% RSLogix 500 project M8017 SEALER OVEN B 20170728 CBP.RSS, saved by version 8.30.00.16 %
PROJECT "M8017"    % processor: MicroLogix 1200 %

PROGRAM FILES
  LAD 2 "MAIN_PROG"  15 rungs
  LAD 4 "INF_XFR_IO"  9 rungs  % InFeed Transfer Input / Output %
  LAD 5 "INF_LOAD"  22 rungs  % InFeed Load Cycle %
  LAD 6 "LANES"  15 rungs  % Lane Conveyor Control %
  LAD 7 "OUT_XFR_IO"  15 rungs  % OutFeed Transfer Input / Output %
  LAD 8 "OUT_UNLOAD"  20 rungs  % OutFeed UnLoad Cycle %
  LAD 10 "FLT"  4 rungs  % Operation Faults %
  LAD 11 "PTV"  8 rungs
  LAD 12 "TOP COAT B"  21 rungs

DATA FILES
  O0 OUTPUT  5 elements
  I1 INPUT  6 elements
  S2 STATUS  66 elements
  B3 BINARY  100 elements
  T4 TIMER  90 elements
  C5 COUNTER  6 elements
  R6 CONTROL  6 elements
  N7 INTEGER  81 elements
  F8 FLOAT  1 elements
  B9 OSR_BIT_2  10 elements  % One Shot Relays and Bit Level 2 %
  B10 HMI  10 elements
  MG11 C8014  1 elements
  T41 TMR_2  100 elements  % Timer Level 2 %
  N71 INT_2  100 elements  % Integer Level 2 %

LADDER 2 "MAIN_PROG"
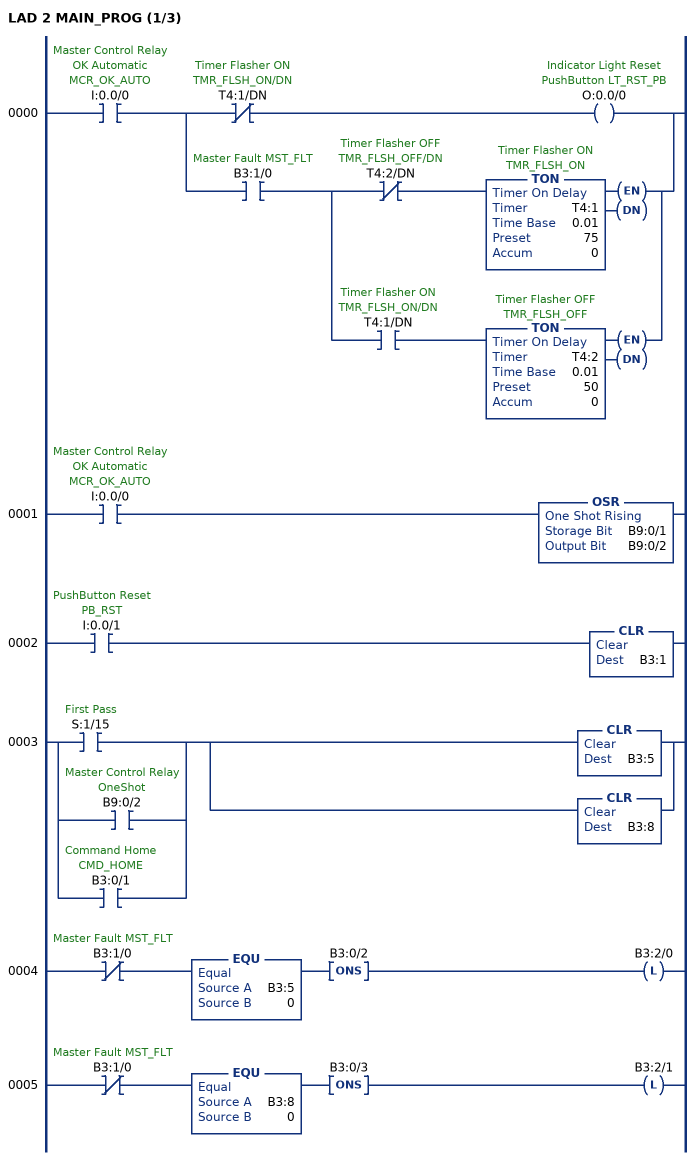
% Rung: 0 %
SOR XIC I:0.0/0 BST XIO T4:1/DN OTE O:0.0/0 NXB XIC B3:1/0 BST XIO T4:2/DN TON T4:1 0.01 75 0 NXB XIC T4:1/DN TON T4:2 0.01 50 0 BND BND EOR
%   I:0.0/0  MCR_OK_AUTO  "Master Control Relay OK Automatic" %
%   T4:1  TMR_FLSH_ON  "Timer Flasher ON" %
%   O:0.0/0  LT_RST_PB  "Indicator Light Reset PushButton" %
%   B3:1/0  MST_FLT  "Master Fault" %
%   T4:2  TMR_FLSH_OFF  "Timer Flasher OFF" %
% Rung: 1 %
SOR XIC I:0.0/0 OSR B9:0/1 B9:0/2 EOR
%   I:0.0/0  MCR_OK_AUTO  "Master Control Relay OK Automatic" %
%   B9:0/2  "Master Control Relay OneShot" %
% Rung: 2 %
SOR XIC I:0.0/1 CLR B3:1 EOR
%   I:0.0/1  PB_RST  "PushButton Reset" %
% Rung: 3 %
SOR BST XIC S:1/15 NXB XIC B9:0/2 NXB XIC B3:0/1 BND BST CLR B3:5 NXB CLR B3:8 BND EOR
%   S:1/15  "First Pass" %
%   B9:0/2  "Master Control Relay OneShot" %
%   B3:0/1  CMD_HOME  "Command Home" %
% Rung: 4 %
SOR XIO B3:1/0 EQU B3:5 0 ONS B3:0/2 OTL B3:2/0 EOR
%   B3:1/0  MST_FLT  "Master Fault" %
% Rung: 5 %
SOR XIO B3:1/0 EQU B3:8 0 ONS B3:0/3 OTL B3:2/1 EOR
%   B3:1/0  MST_FLT  "Master Fault" %

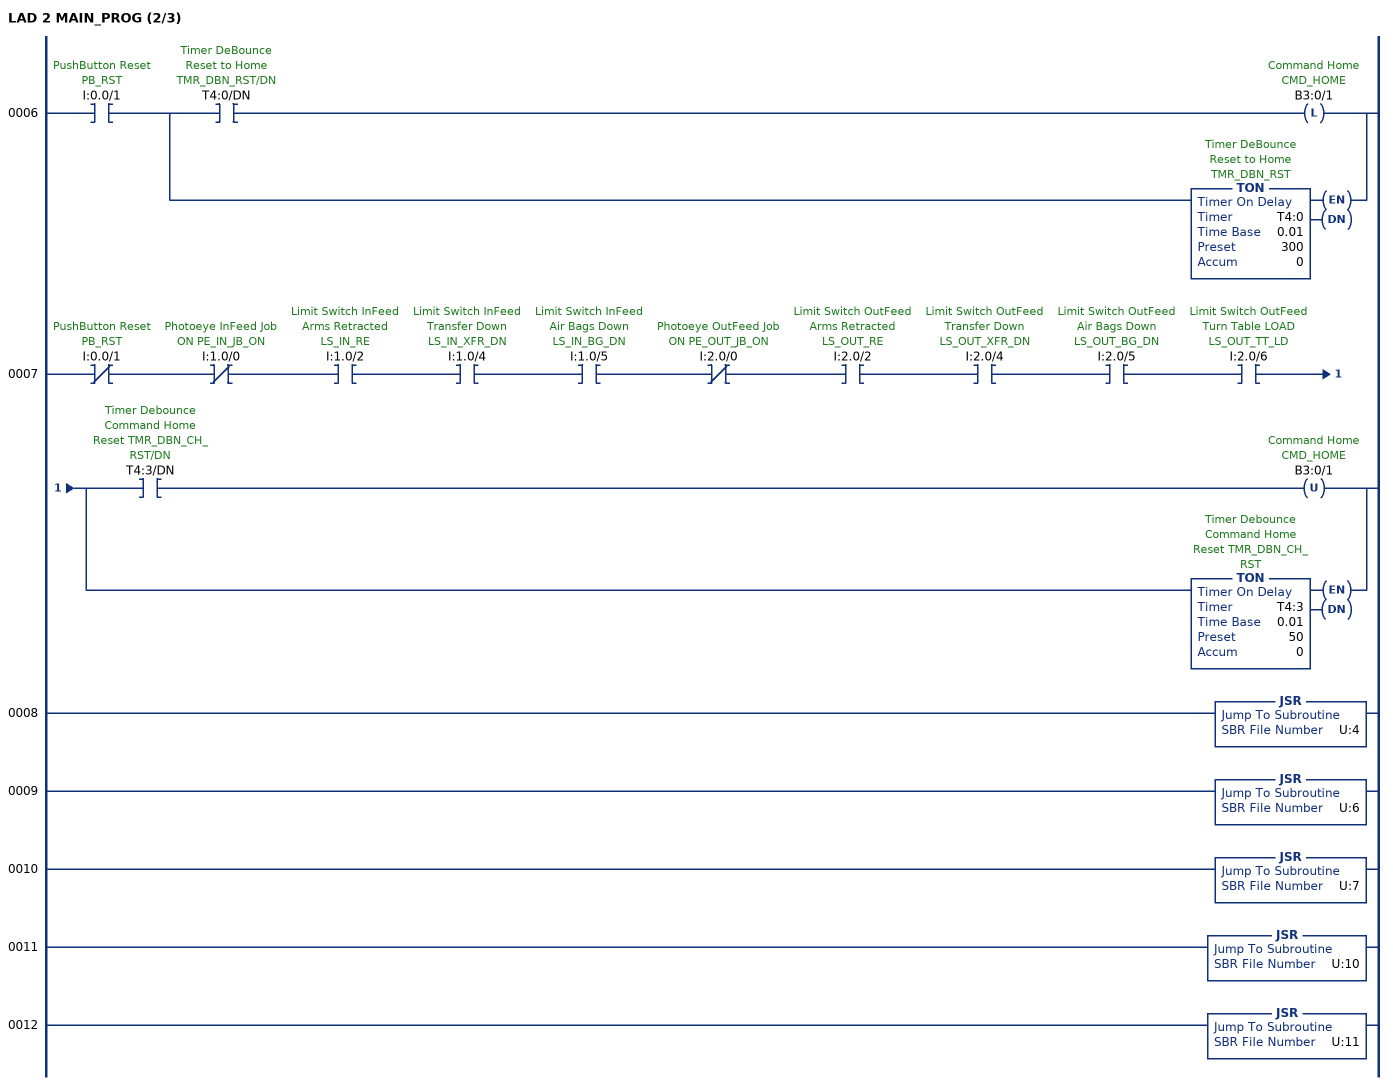
% Rung: 6 %
SOR XIC I:0.0/1 BST XIC T4:0/DN OTL B3:0/1 NXB TON T4:0 0.01 300 0 BND EOR
%   I:0.0/1  PB_RST  "PushButton Reset" %
%   T4:0  TMR_DBN_RST  "Timer DeBounce Reset to Home" %
%   B3:0/1  CMD_HOME  "Command Home" %
% Rung: 7 %
SOR XIO I:0.0/1 XIO I:1.0/0 XIC I:1.0/2 XIC I:1.0/4 XIC I:1.0/5 XIO I:2.0/0 XIC I:2.0/2 XIC I:2.0/4 XIC I:2.0/5 XIC I:2.0/6 BST XIC T4:3/DN OTU B3:0/1 NXB TON T4:3 0.01 50 0 BND EOR
%   I:0.0/1  PB_RST  "PushButton Reset" %
%   I:1.0/0  PE_IN_JB_ON  "Photoeye InFeed Job ON" %
%   I:1.0/2  LS_IN_RE  "Limit Switch InFeed Arms Retracted" %
%   I:1.0/4  LS_IN_XFR_DN  "Limit Switch InFeed Transfer Down" %
%   I:1.0/5  LS_IN_BG_DN  "Limit Switch InFeed Air Bags Down" %
%   I:2.0/0  PE_OUT_JB_ON  "Photoeye OutFeed Job ON" %
%   I:2.0/2  LS_OUT_RE  "Limit Switch OutFeed Arms Retracted" %
%   I:2.0/4  LS_OUT_XFR_DN  "Limit Switch OutFeed Transfer Down" %
%   I:2.0/5  LS_OUT_BG_DN  "Limit Switch OutFeed Air Bags Down" %
%   I:2.0/6  LS_OUT_TT_LD  "Limit Switch OutFeed Turn Table LOAD" %
%   T4:3  TMR_DBN_CH_RST  "Timer Debounce Command Home Reset" %
%   B3:0/1  CMD_HOME  "Command Home" %
% Rung: 8 %
SOR JSR U:4 EOR
% Rung: 9 %
SOR JSR U:6 EOR
% Rung: 10 %
SOR JSR U:7 EOR
% Rung: 11 %
SOR JSR U:10 EOR
% Rung: 12 %
SOR JSR U:11 EOR

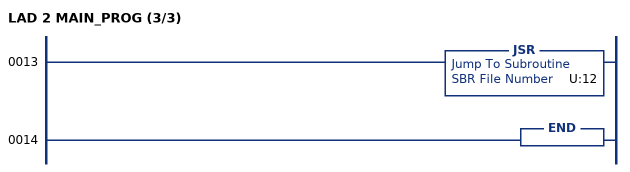
% Rung: 13 %
SOR JSR U:12 EOR
% Rung: 14 %
SOR END EOR

LADDER 4 "INF_XFR_IO"    % InFeed Transfer Input / Output %
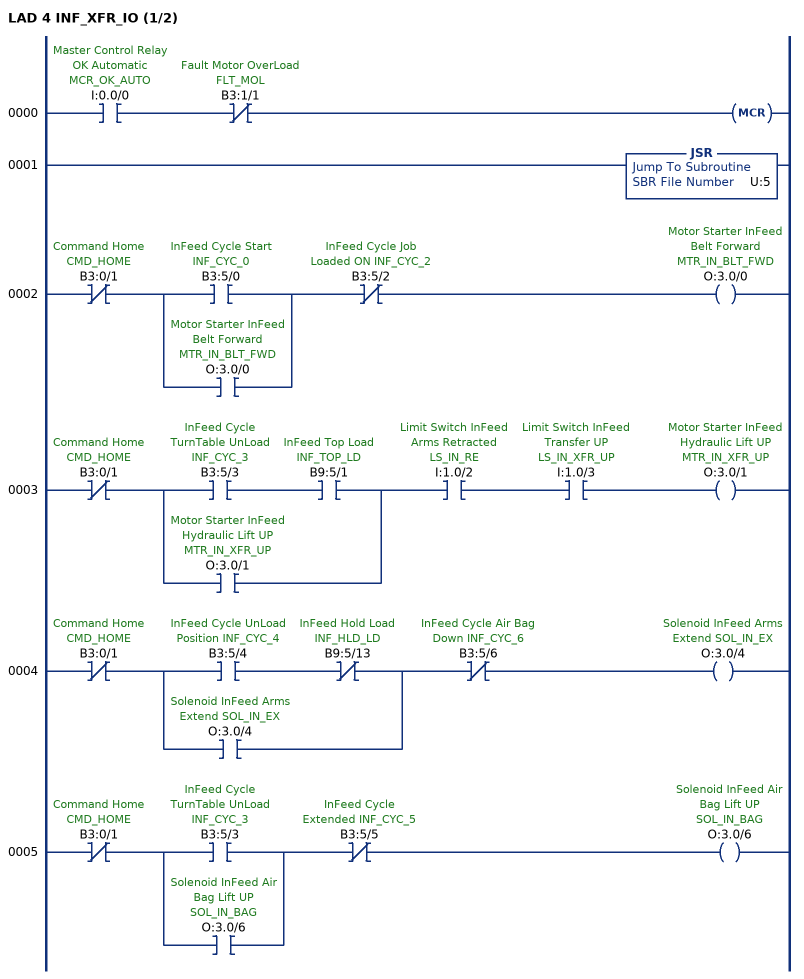
% Rung: 0 %
SOR XIC I:0.0/0 XIO B3:1/1 MCR EOR
%   I:0.0/0  MCR_OK_AUTO  "Master Control Relay OK Automatic" %
%   B3:1/1  FLT_MOL  "Fault Motor OverLoad" %
% Rung: 1 %
SOR JSR U:5 EOR
% Rung: 2 %  % edit flag set %
SOR XIO B3:0/1 BST XIC B3:5/0 NXB XIC O:3.0/0 BND XIO B3:5/2 OTE O:3.0/0 EOR
%   B3:0/1  CMD_HOME  "Command Home" %
%   B3:5/0  INF_CYC_0  "InFeed Cycle Start" %
%   O:3.0/0  MTR_IN_BLT_FWD  "Motor Starter InFeed Belt Forward" %
%   B3:5/2  INF_CYC_2  "InFeed Cycle Job Loaded ON" %
% Rung: 3 %
SOR XIO B3:0/1 BST XIC B3:5/3 XIC B9:5/1 NXB XIC O:3.0/1 BND XIC I:1.0/2 XIC I:1.0/3 OTE O:3.0/1 EOR
%   B3:0/1  CMD_HOME  "Command Home" %
%   B3:5/3  INF_CYC_3  "InFeed Cycle TurnTable UnLoad" %
%   B9:5/1  INF_TOP_LD  "InFeed Top Load" %
%   O:3.0/1  MTR_IN_XFR_UP  "Motor Starter InFeed Hydraulic Lift UP" %
%   I:1.0/2  LS_IN_RE  "Limit Switch InFeed Arms Retracted" %
%   I:1.0/3  LS_IN_XFR_UP  "Limit Switch InFeed Transfer UP" %
% Rung: 4 %
SOR XIO B3:0/1 BST XIC B3:5/4 XIO B9:5/13 NXB XIC O:3.0/4 BND XIO B3:5/6 OTE O:3.0/4 EOR
%   B3:0/1  CMD_HOME  "Command Home" %
%   B3:5/4  INF_CYC_4  "InFeed Cycle UnLoad Position" %
%   B9:5/13  INF_HLD_LD  "InFeed Hold Load" %
%   O:3.0/4  SOL_IN_EX  "Solenoid InFeed Arms Extend" %
%   B3:5/6  INF_CYC_6  "InFeed Cycle Air Bag Down" %
% Rung: 5 %
SOR XIO B3:0/1 BST XIC B3:5/3 NXB XIC O:3.0/6 BND XIO B3:5/5 OTE O:3.0/6 EOR
%   B3:0/1  CMD_HOME  "Command Home" %
%   B3:5/3  INF_CYC_3  "InFeed Cycle TurnTable UnLoad" %
%   O:3.0/6  SOL_IN_BAG  "Solenoid InFeed Air Bag Lift UP" %
%   B3:5/5  INF_CYC_5  "InFeed Cycle Extended" %

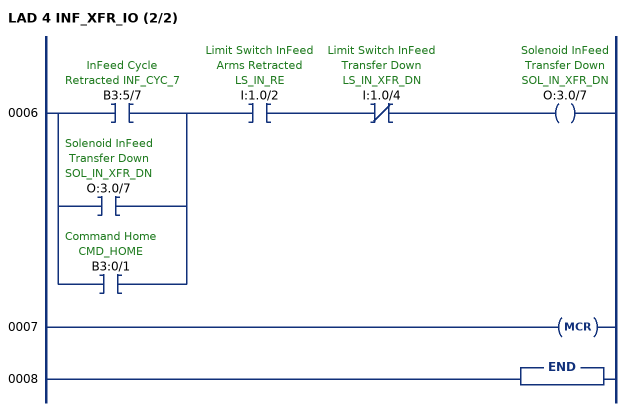
% Rung: 6 %
SOR BST XIC B3:5/7 NXB XIC O:3.0/7 NXB XIC B3:0/1 BND XIC I:1.0/2 XIO I:1.0/4 OTE O:3.0/7 EOR
%   B3:5/7  INF_CYC_7  "InFeed Cycle Retracted" %
%   O:3.0/7  SOL_IN_XFR_DN  "Solenoid InFeed Transfer Down" %
%   B3:0/1  CMD_HOME  "Command Home" %
%   I:1.0/2  LS_IN_RE  "Limit Switch InFeed Arms Retracted" %
%   I:1.0/4  LS_IN_XFR_DN  "Limit Switch InFeed Transfer Down" %
% Rung: 7 %
SOR MCR EOR
% Rung: 8 %
SOR END EOR

LADDER 5 "INF_LOAD"    % InFeed Load Cycle %
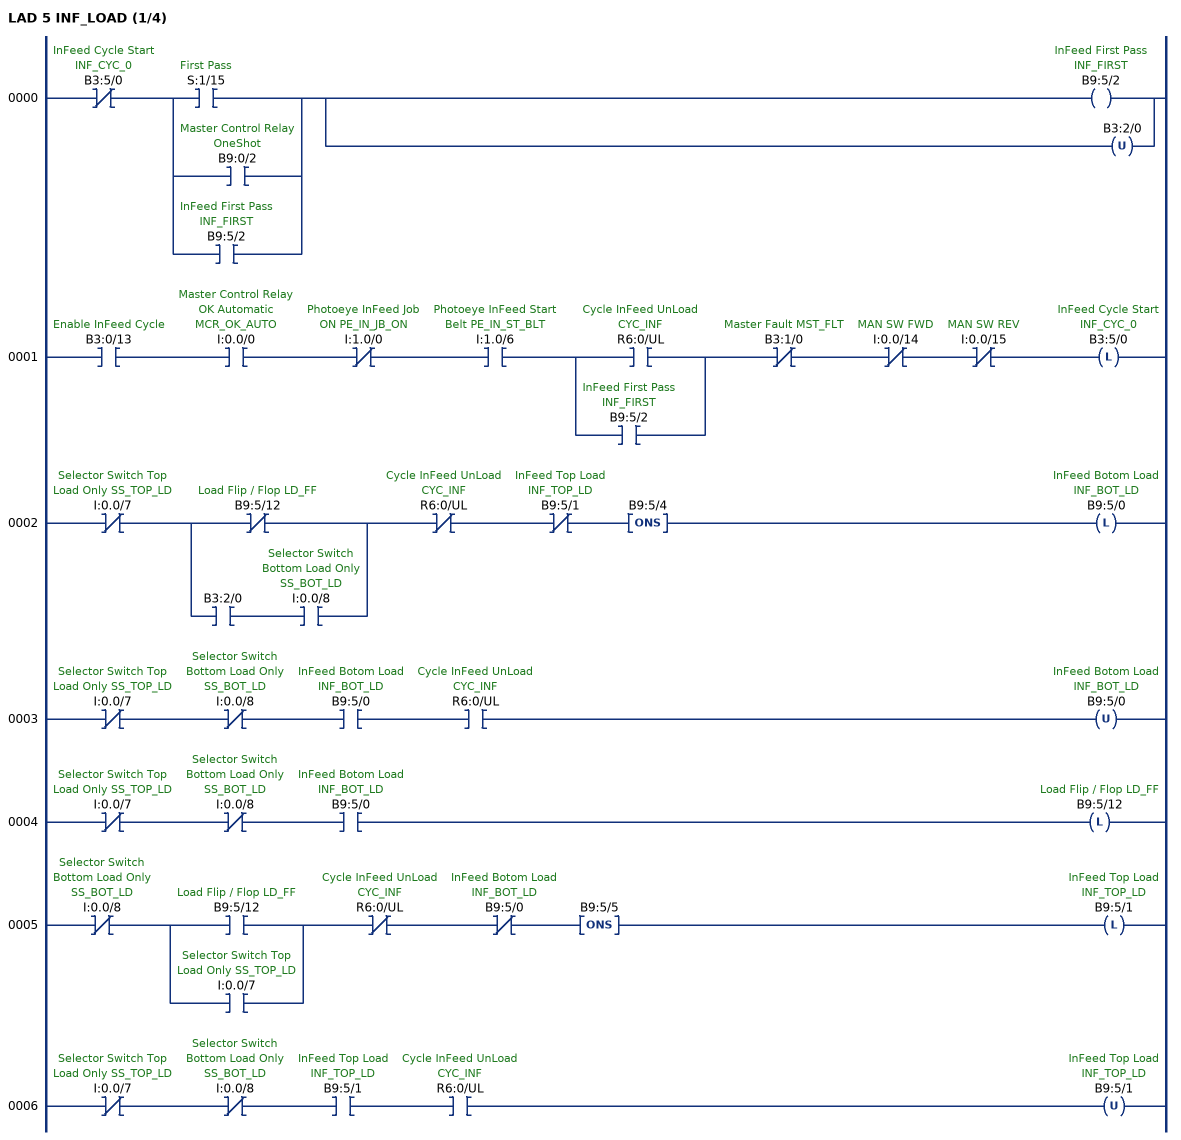
% Rung: 0 %
SOR XIO B3:5/0 BST XIC S:1/15 NXB XIC B9:0/2 NXB XIC B9:5/2 BND BST OTE B9:5/2 NXB OTU B3:2/0 BND EOR
%   B3:5/0  INF_CYC_0  "InFeed Cycle Start" %
%   S:1/15  "First Pass" %
%   B9:0/2  "Master Control Relay OneShot" %
%   B9:5/2  INF_FIRST  "InFeed First Pass" %
% Rung: 1 %  % edit flag set %
SOR XIC B3:0/13 XIC I:0.0/0 XIO I:1.0/0 XIC I:1.0/6 BST XIC R6:0/UL NXB XIC B9:5/2 BND XIO B3:1/0 XIO I:0.0/14 XIO I:0.0/15 OTL B3:5/0 EOR
%   B3:0/13  "Enable InFeed Cycle" %
%   I:0.0/0  MCR_OK_AUTO  "Master Control Relay OK Automatic" %
%   I:1.0/0  PE_IN_JB_ON  "Photoeye InFeed Job ON" %
%   I:1.0/6  PE_IN_ST_BLT  "Photoeye InFeed Start Belt" %
%   R6:0/UL  CYC_INF  "Cycle InFeed UnLoad" %
%   B9:5/2  INF_FIRST  "InFeed First Pass" %
%   B3:1/0  MST_FLT  "Master Fault" %
%   I:0.0/14  "MAN SW FWD" %
%   I:0.0/15  "MAN SW REV" %
%   B3:5/0  INF_CYC_0  "InFeed Cycle Start" %
% Rung: 2 %
SOR XIO I:0.0/7 BST XIO B9:5/12 NXB XIC B3:2/0 XIC I:0.0/8 BND XIO R6:0/UL XIO B9:5/1 ONS B9:5/4 OTL B9:5/0 EOR
%   I:0.0/7  SS_TOP_LD  "Selector Switch Top Load Only" %
%   B9:5/12  LD_FF  "Load Flip / Flop" %
%   I:0.0/8  SS_BOT_LD  "Selector Switch Bottom Load Only" %
%   R6:0/UL  CYC_INF  "Cycle InFeed UnLoad" %
%   B9:5/1  INF_TOP_LD  "InFeed Top Load" %
%   B9:5/0  INF_BOT_LD  "InFeed Botom Load" %
% Rung: 3 %
SOR XIO I:0.0/7 XIO I:0.0/8 XIC B9:5/0 XIC R6:0/UL OTU B9:5/0 EOR
%   I:0.0/7  SS_TOP_LD  "Selector Switch Top Load Only" %
%   I:0.0/8  SS_BOT_LD  "Selector Switch Bottom Load Only" %
%   B9:5/0  INF_BOT_LD  "InFeed Botom Load" %
%   R6:0/UL  CYC_INF  "Cycle InFeed UnLoad" %
% Rung: 4 %
SOR XIO I:0.0/7 XIO I:0.0/8 XIC B9:5/0 OTL B9:5/12 EOR
%   I:0.0/7  SS_TOP_LD  "Selector Switch Top Load Only" %
%   I:0.0/8  SS_BOT_LD  "Selector Switch Bottom Load Only" %
%   B9:5/0  INF_BOT_LD  "InFeed Botom Load" %
%   B9:5/12  LD_FF  "Load Flip / Flop" %
% Rung: 5 %
SOR XIO I:0.0/8 BST XIC B9:5/12 NXB XIC I:0.0/7 BND XIO R6:0/UL XIO B9:5/0 ONS B9:5/5 OTL B9:5/1 EOR
%   I:0.0/8  SS_BOT_LD  "Selector Switch Bottom Load Only" %
%   B9:5/12  LD_FF  "Load Flip / Flop" %
%   I:0.0/7  SS_TOP_LD  "Selector Switch Top Load Only" %
%   R6:0/UL  CYC_INF  "Cycle InFeed UnLoad" %
%   B9:5/0  INF_BOT_LD  "InFeed Botom Load" %
%   B9:5/1  INF_TOP_LD  "InFeed Top Load" %
% Rung: 6 %
SOR XIO I:0.0/7 XIO I:0.0/8 XIC B9:5/1 XIC R6:0/UL OTU B9:5/1 EOR
%   I:0.0/7  SS_TOP_LD  "Selector Switch Top Load Only" %
%   I:0.0/8  SS_BOT_LD  "Selector Switch Bottom Load Only" %
%   B9:5/1  INF_TOP_LD  "InFeed Top Load" %
%   R6:0/UL  CYC_INF  "Cycle InFeed UnLoad" %

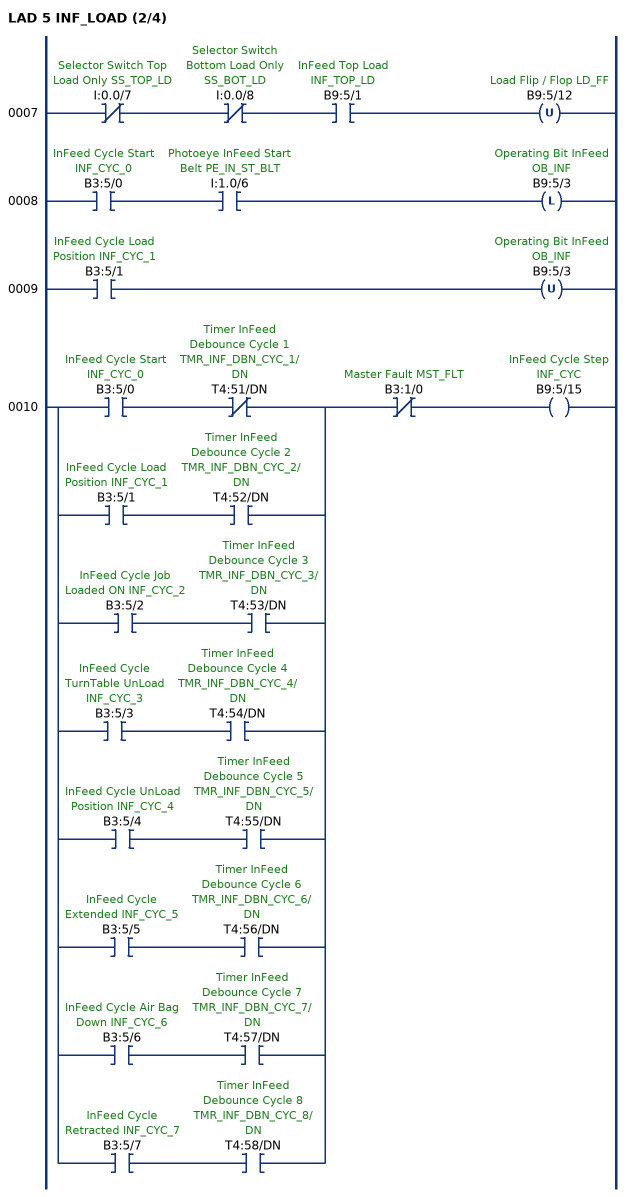
% Rung: 7 %
SOR XIO I:0.0/7 XIO I:0.0/8 XIC B9:5/1 OTU B9:5/12 EOR
%   I:0.0/7  SS_TOP_LD  "Selector Switch Top Load Only" %
%   I:0.0/8  SS_BOT_LD  "Selector Switch Bottom Load Only" %
%   B9:5/1  INF_TOP_LD  "InFeed Top Load" %
%   B9:5/12  LD_FF  "Load Flip / Flop" %
% Rung: 8 %
SOR XIC B3:5/0 XIC I:1.0/6 OTL B9:5/3 EOR
%   B3:5/0  INF_CYC_0  "InFeed Cycle Start" %
%   I:1.0/6  PE_IN_ST_BLT  "Photoeye InFeed Start Belt" %
%   B9:5/3  OB_INF  "Operating Bit InFeed" %
% Rung: 9 %
SOR XIC B3:5/1 OTU B9:5/3 EOR
%   B3:5/1  INF_CYC_1  "InFeed Cycle Load Position" %
%   B9:5/3  OB_INF  "Operating Bit InFeed" %
% Rung: 10 %
SOR BST XIC B3:5/0 XIO T4:51/DN NXB XIC B3:5/1 XIC T4:52/DN NXB XIC B3:5/2 XIC T4:53/DN NXB XIC B3:5/3 XIC T4:54/DN NXB XIC B3:5/4 XIC T4:55/DN NXB XIC B3:5/5 XIC T4:56/DN NXB XIC B3:5/6 XIC T4:57/DN NXB XIC B3:5/7 XIC T4:58/DN BND XIO B3:1/0 OTE B9:5/15 EOR
%   B3:5/0  INF_CYC_0  "InFeed Cycle Start" %
%   T4:51  TMR_INF_DBN_CYC_1  "Timer InFeed Debounce Cycle 1" %
%   B3:5/1  INF_CYC_1  "InFeed Cycle Load Position" %
%   T4:52  TMR_INF_DBN_CYC_2  "Timer InFeed Debounce Cycle 2" %
%   B3:5/2  INF_CYC_2  "InFeed Cycle Job Loaded ON" %
%   T4:53  TMR_INF_DBN_CYC_3  "Timer InFeed Debounce Cycle 3" %
%   B3:5/3  INF_CYC_3  "InFeed Cycle TurnTable UnLoad" %
%   T4:54  TMR_INF_DBN_CYC_4  "Timer InFeed Debounce Cycle 4" %
%   B3:5/4  INF_CYC_4  "InFeed Cycle UnLoad Position" %
%   T4:55  TMR_INF_DBN_CYC_5  "Timer InFeed Debounce Cycle 5" %
%   B3:5/5  INF_CYC_5  "InFeed Cycle Extended" %
%   T4:56  TMR_INF_DBN_CYC_6  "Timer InFeed Debounce Cycle 6" %
%   B3:5/6  INF_CYC_6  "InFeed Cycle Air Bag Down" %
%   T4:57  TMR_INF_DBN_CYC_7  "Timer InFeed Debounce Cycle 7" %
%   B3:5/7  INF_CYC_7  "InFeed Cycle Retracted" %
%   T4:58  TMR_INF_DBN_CYC_8  "Timer InFeed Debounce Cycle 8" %
%   B3:1/0  MST_FLT  "Master Fault" %
%   B9:5/15  INF_CYC  "InFeed Cycle Step" %

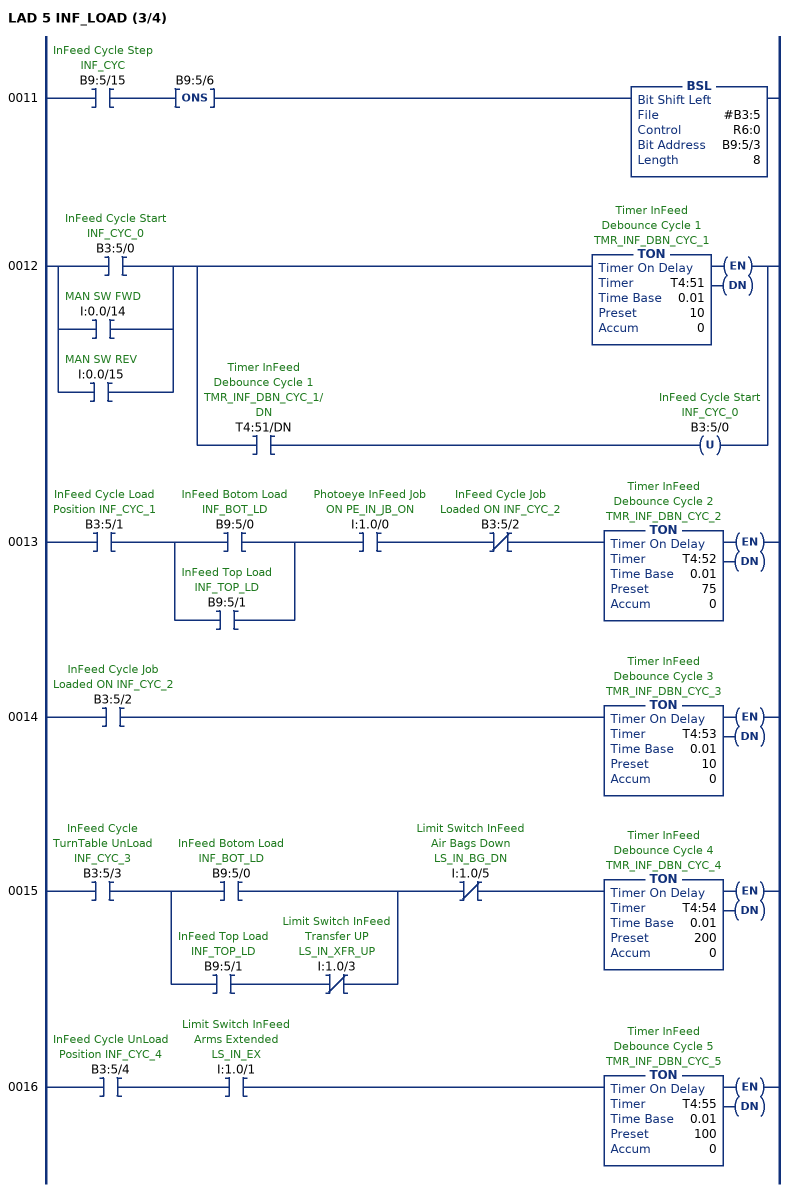
% Rung: 11 %
SOR XIC B9:5/15 ONS B9:5/6 BSL #B3:5 R6:0 B9:5/3 8 EOR
%   B9:5/15  INF_CYC  "InFeed Cycle Step" %
%   R6:0  "Cycle InFeed" %
%   B9:5/3  OB_INF  "Operating Bit InFeed" %
% Rung: 12 %  % edit flag set %
SOR BST XIC B3:5/0 NXB XIC I:0.0/14 NXB XIC I:0.0/15 BND BST TON T4:51 0.01 10 0 NXB XIC T4:51/DN OTU B3:5/0 BND EOR
%   B3:5/0  INF_CYC_0  "InFeed Cycle Start" %
%   I:0.0/14  "MAN SW FWD" %
%   I:0.0/15  "MAN SW REV" %
%   T4:51  TMR_INF_DBN_CYC_1  "Timer InFeed Debounce Cycle 1" %
% Rung: 13 %
SOR XIC B3:5/1 BST XIC B9:5/0 NXB XIC B9:5/1 BND XIC I:1.0/0 XIO B3:5/2 TON T4:52 0.01 75 0 EOR
%   B3:5/1  INF_CYC_1  "InFeed Cycle Load Position" %
%   B9:5/0  INF_BOT_LD  "InFeed Botom Load" %
%   B9:5/1  INF_TOP_LD  "InFeed Top Load" %
%   I:1.0/0  PE_IN_JB_ON  "Photoeye InFeed Job ON" %
%   B3:5/2  INF_CYC_2  "InFeed Cycle Job Loaded ON" %
%   T4:52  TMR_INF_DBN_CYC_2  "Timer InFeed Debounce Cycle 2" %
% Rung: 14 %
SOR XIC B3:5/2 TON T4:53 0.01 10 0 EOR
%   B3:5/2  INF_CYC_2  "InFeed Cycle Job Loaded ON" %
%   T4:53  TMR_INF_DBN_CYC_3  "Timer InFeed Debounce Cycle 3" %
% Rung: 15 %
SOR XIC B3:5/3 BST XIC B9:5/0 NXB XIC B9:5/1 XIO I:1.0/3 BND XIO I:1.0/5 TON T4:54 0.01 200 0 EOR
%   B3:5/3  INF_CYC_3  "InFeed Cycle TurnTable UnLoad" %
%   B9:5/0  INF_BOT_LD  "InFeed Botom Load" %
%   B9:5/1  INF_TOP_LD  "InFeed Top Load" %
%   I:1.0/3  LS_IN_XFR_UP  "Limit Switch InFeed Transfer UP" %
%   I:1.0/5  LS_IN_BG_DN  "Limit Switch InFeed Air Bags Down" %
%   T4:54  TMR_INF_DBN_CYC_4  "Timer InFeed Debounce Cycle 4" %
% Rung: 16 %
SOR XIC B3:5/4 XIC I:1.0/1 TON T4:55 0.01 100 0 EOR
%   B3:5/4  INF_CYC_4  "InFeed Cycle UnLoad Position" %
%   I:1.0/1  LS_IN_EX  "Limit Switch InFeed Arms Extended" %
%   T4:55  TMR_INF_DBN_CYC_5  "Timer InFeed Debounce Cycle 5" %

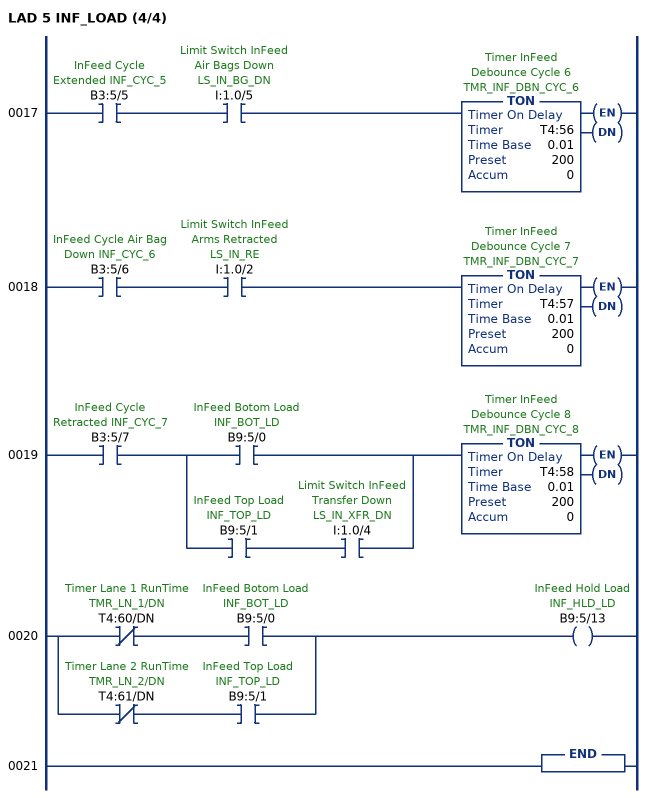
% Rung: 17 %
SOR XIC B3:5/5 XIC I:1.0/5 TON T4:56 0.01 200 0 EOR
%   B3:5/5  INF_CYC_5  "InFeed Cycle Extended" %
%   I:1.0/5  LS_IN_BG_DN  "Limit Switch InFeed Air Bags Down" %
%   T4:56  TMR_INF_DBN_CYC_6  "Timer InFeed Debounce Cycle 6" %
% Rung: 18 %
SOR XIC B3:5/6 XIC I:1.0/2 TON T4:57 0.01 200 0 EOR
%   B3:5/6  INF_CYC_6  "InFeed Cycle Air Bag Down" %
%   I:1.0/2  LS_IN_RE  "Limit Switch InFeed Arms Retracted" %
%   T4:57  TMR_INF_DBN_CYC_7  "Timer InFeed Debounce Cycle 7" %
% Rung: 19 %
SOR XIC B3:5/7 BST XIC B9:5/0 NXB XIC B9:5/1 XIC I:1.0/4 BND TON T4:58 0.01 200 0 EOR
%   B3:5/7  INF_CYC_7  "InFeed Cycle Retracted" %
%   B9:5/0  INF_BOT_LD  "InFeed Botom Load" %
%   B9:5/1  INF_TOP_LD  "InFeed Top Load" %
%   I:1.0/4  LS_IN_XFR_DN  "Limit Switch InFeed Transfer Down" %
%   T4:58  TMR_INF_DBN_CYC_8  "Timer InFeed Debounce Cycle 8" %
% Rung: 20 %
SOR BST XIO T4:60/DN XIC B9:5/0 NXB XIO T4:61/DN XIC B9:5/1 BND OTE B9:5/13 EOR
%   T4:60  TMR_LN_1  "Timer Lane 1 RunTime" %
%   B9:5/0  INF_BOT_LD  "InFeed Botom Load" %
%   T4:61  TMR_LN_2  "Timer Lane 2 RunTime" %
%   B9:5/1  INF_TOP_LD  "InFeed Top Load" %
%   B9:5/13  INF_HLD_LD  "InFeed Hold Load" %
% Rung: 21 %
SOR END EOR

LADDER 6 "LANES"    % Lane Conveyor Control %
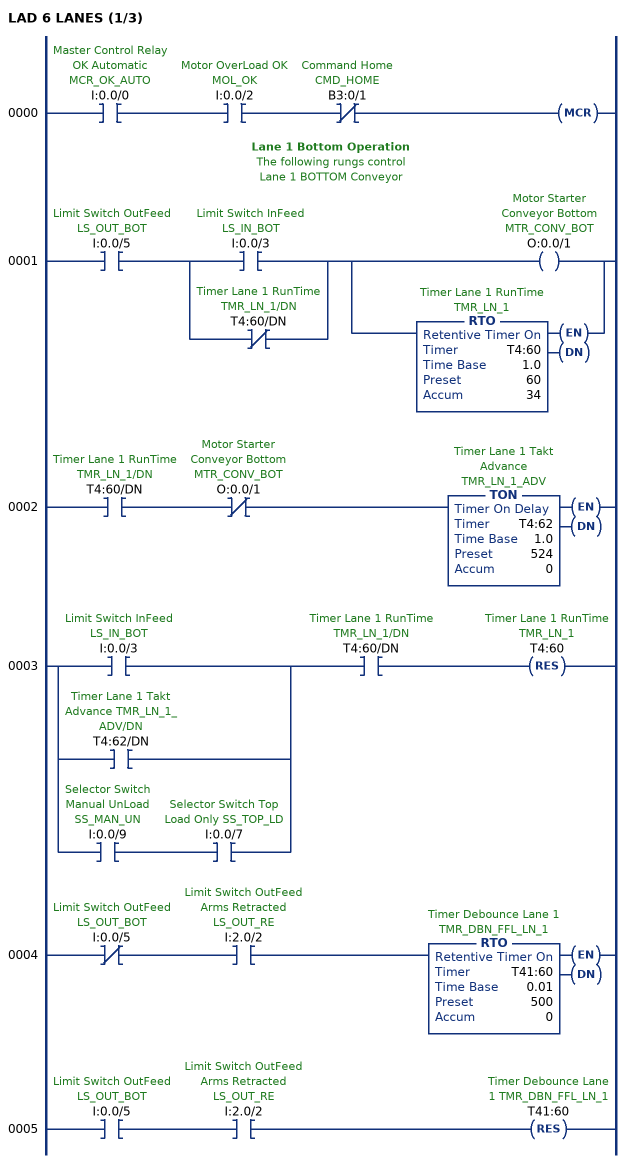
% Rung: 0 %
SOR XIC I:0.0/0 XIC I:0.0/2 XIO B3:0/1 MCR EOR
%   I:0.0/0  MCR_OK_AUTO  "Master Control Relay OK Automatic" %
%   I:0.0/2  MOL_OK  "Motor OverLoad OK" %
%   B3:0/1  CMD_HOME  "Command Home" %
% Rung: 1 %
% TITLE: Lane 1 Bottom Operation %
% The following rungs control
% Lane 1 BOTTOM Conveyor %
SOR XIC I:0.0/5 BST XIC I:0.0/3 NXB XIO T4:60/DN BND BST OTE O:0.0/1 NXB RTO T4:60 1.0 60 34 BND EOR
%   I:0.0/5  LS_OUT_BOT  "Limit Switch OutFeed" %
%   I:0.0/3  LS_IN_BOT  "Limit Switch InFeed" %
%   T4:60  TMR_LN_1  "Timer Lane 1 RunTime" %
%   O:0.0/1  MTR_CONV_BOT  "Motor Starter Conveyor Bottom" %
% Rung: 2 %  % edit flag set %
SOR XIC T4:60/DN XIO O:0.0/1 TON T4:62 1.0 524 0 EOR
%   T4:60  TMR_LN_1  "Timer Lane 1 RunTime" %
%   O:0.0/1  MTR_CONV_BOT  "Motor Starter Conveyor Bottom" %
%   T4:62  TMR_LN_1_ADV  "Timer Lane 1 Takt Advance" %
% Rung: 3 %
SOR BST XIC I:0.0/3 NXB XIC T4:62/DN NXB XIC I:0.0/9 XIC I:0.0/7 BND XIC T4:60/DN RES T4:60 EOR
%   I:0.0/3  LS_IN_BOT  "Limit Switch InFeed" %
%   T4:62  TMR_LN_1_ADV  "Timer Lane 1 Takt Advance" %
%   I:0.0/9  SS_MAN_UN  "Selector Switch Manual UnLoad" %
%   I:0.0/7  SS_TOP_LD  "Selector Switch Top Load Only" %
%   T4:60  TMR_LN_1  "Timer Lane 1 RunTime" %
% Rung: 4 %
SOR XIO I:0.0/5 XIC I:2.0/2 RTO T41:60 0.01 500 0 EOR
%   I:0.0/5  LS_OUT_BOT  "Limit Switch OutFeed" %
%   I:2.0/2  LS_OUT_RE  "Limit Switch OutFeed Arms Retracted" %
%   T41:60  TMR_DBN_FFL_LN_1  "Timer Debounce Lane 1" %
% Rung: 5 %
SOR XIC I:0.0/5 XIC I:2.0/2 RES T41:60 EOR
%   I:0.0/5  LS_OUT_BOT  "Limit Switch OutFeed" %
%   I:2.0/2  LS_OUT_RE  "Limit Switch OutFeed Arms Retracted" %
%   T41:60  TMR_DBN_FFL_LN_1  "Timer Debounce Lane 1" %

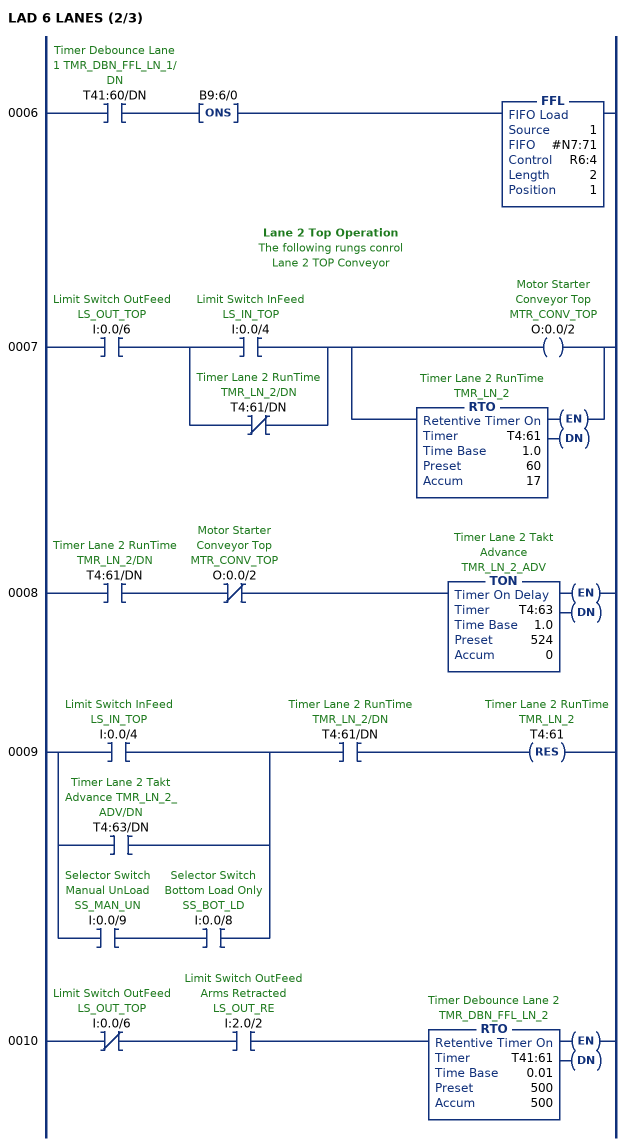
% Rung: 6 %
SOR XIC T41:60/DN ONS B9:6/0 FFL 1 #N7:71 R6:4 2 1 EOR
%   T41:60  TMR_DBN_FFL_LN_1  "Timer Debounce Lane 1" %
%   N7:71  OUT_FIFO_1  "OutFeed FIFO Buffer Position 1" %
%   R6:4  "InFeed FIFO Stack Control" %
% Rung: 7 %
% TITLE: Lane 2 Top Operation %
% The following rungs conrol
% Lane 2 TOP Conveyor %
SOR XIC I:0.0/6 BST XIC I:0.0/4 NXB XIO T4:61/DN BND BST OTE O:0.0/2 NXB RTO T4:61 1.0 60 17 BND EOR
%   I:0.0/6  LS_OUT_TOP  "Limit Switch OutFeed" %
%   I:0.0/4  LS_IN_TOP  "Limit Switch InFeed" %
%   T4:61  TMR_LN_2  "Timer Lane 2 RunTime" %
%   O:0.0/2  MTR_CONV_TOP  "Motor Starter Conveyor Top" %
% Rung: 8 %  % edit flag set %
SOR XIC T4:61/DN XIO O:0.0/2 TON T4:63 1.0 524 0 EOR
%   T4:61  TMR_LN_2  "Timer Lane 2 RunTime" %
%   O:0.0/2  MTR_CONV_TOP  "Motor Starter Conveyor Top" %
%   T4:63  TMR_LN_2_ADV  "Timer Lane 2 Takt Advance" %
% Rung: 9 %
SOR BST XIC I:0.0/4 NXB XIC T4:63/DN NXB XIC I:0.0/9 XIC I:0.0/8 BND XIC T4:61/DN RES T4:61 EOR
%   I:0.0/4  LS_IN_TOP  "Limit Switch InFeed" %
%   T4:63  TMR_LN_2_ADV  "Timer Lane 2 Takt Advance" %
%   I:0.0/9  SS_MAN_UN  "Selector Switch Manual UnLoad" %
%   I:0.0/8  SS_BOT_LD  "Selector Switch Bottom Load Only" %
%   T4:61  TMR_LN_2  "Timer Lane 2 RunTime" %
% Rung: 10 %
SOR XIO I:0.0/6 XIC I:2.0/2 RTO T41:61 0.01 500 500 EOR
%   I:0.0/6  LS_OUT_TOP  "Limit Switch OutFeed" %
%   I:2.0/2  LS_OUT_RE  "Limit Switch OutFeed Arms Retracted" %
%   T41:61  TMR_DBN_FFL_LN_2  "Timer Debounce Lane 2" %

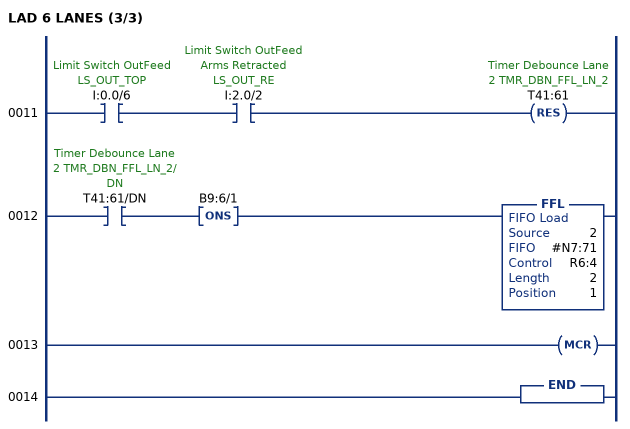
% Rung: 11 %
SOR XIC I:0.0/6 XIC I:2.0/2 RES T41:61 EOR
%   I:0.0/6  LS_OUT_TOP  "Limit Switch OutFeed" %
%   I:2.0/2  LS_OUT_RE  "Limit Switch OutFeed Arms Retracted" %
%   T41:61  TMR_DBN_FFL_LN_2  "Timer Debounce Lane 2" %
% Rung: 12 %
SOR XIC T41:61/DN ONS B9:6/1 FFL 2 #N7:71 R6:4 2 1 EOR
%   T41:61  TMR_DBN_FFL_LN_2  "Timer Debounce Lane 2" %
%   N7:71  OUT_FIFO_1  "OutFeed FIFO Buffer Position 1" %
%   R6:4  "InFeed FIFO Stack Control" %
% Rung: 13 %
SOR MCR EOR
% Rung: 14 %
SOR END EOR

LADDER 7 "OUT_XFR_IO"    % OutFeed Transfer Input / Output %
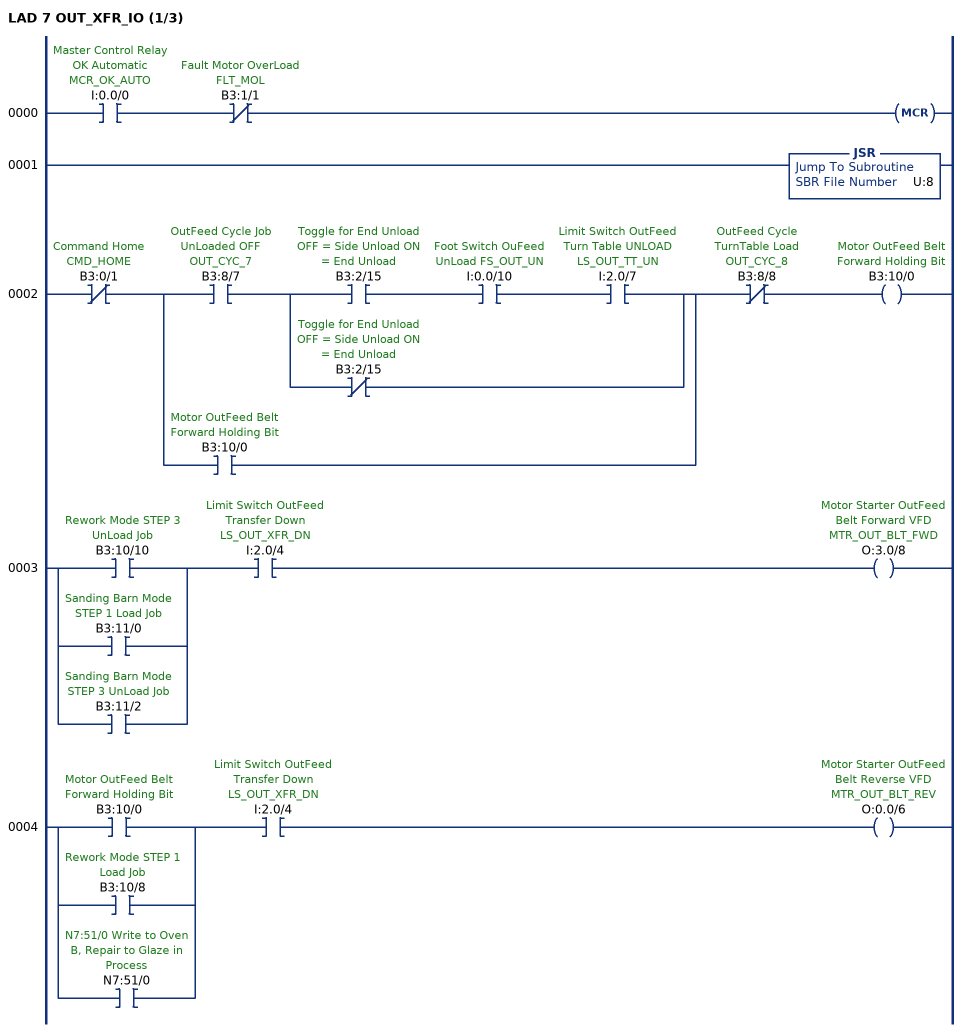
% Rung: 0 %
SOR XIC I:0.0/0 XIO B3:1/1 MCR EOR
%   I:0.0/0  MCR_OK_AUTO  "Master Control Relay OK Automatic" %
%   B3:1/1  FLT_MOL  "Fault Motor OverLoad" %
% Rung: 1 %
SOR JSR U:8 EOR
% Rung: 2 %
SOR XIO B3:0/1 BST XIC B3:8/7 BST XIC B3:2/15 XIC I:0.0/10 XIC I:2.0/7 NXB XIO B3:2/15 BND NXB XIC B3:10/0 BND XIO B3:8/8 OTE B3:10/0 EOR
%   B3:0/1  CMD_HOME  "Command Home" %
%   B3:8/7  OUT_CYC_7  "OutFeed Cycle Job UnLoaded OFF" %
%   B3:2/15  "Toggle for End Unload OFF = Side Unload ON = End Unload" %
%   I:0.0/10  FS_OUT_UN  "Foot Switch OuFeed UnLoad" %
%   I:2.0/7  LS_OUT_TT_UN  "Limit Switch OutFeed Turn Table UNLOAD" %
%   B3:10/0  "Motor OutFeed Belt Forward Holding Bit" %
%   B3:8/8  OUT_CYC_8  "OutFeed Cycle TurnTable Load" %
% Rung: 3 %  % edit flag set %
SOR BST XIC B3:10/10 NXB XIC B3:11/0 NXB XIC B3:11/2 BND XIC I:2.0/4 OTE O:3.0/8 EOR
%   B3:10/10  "Rework Mode STEP 3 UnLoad Job" %
%   B3:11/0  "Sanding Barn Mode STEP 1 Load Job" %
%   B3:11/2  "Sanding Barn Mode STEP 3 UnLoad Job" %
%   I:2.0/4  LS_OUT_XFR_DN  "Limit Switch OutFeed Transfer Down" %
%   O:3.0/8  MTR_OUT_BLT_FWD  "Motor Starter OutFeed Belt Forward VFD" %
% Rung: 4 %  % edit flag set %
SOR BST XIC B3:10/0 NXB XIC B3:10/8 NXB XIC N7:51/0 BND XIC I:2.0/4 OTE O:0.0/6 EOR
%   B3:10/0  "Motor OutFeed Belt Forward Holding Bit" %
%   B3:10/8  "Rework Mode STEP 1 Load Job" %
%   N7:51/0  "N7:51/0 Write to Oven B, Repair to Glaze in Process" %
%   I:2.0/4  LS_OUT_XFR_DN  "Limit Switch OutFeed Transfer Down" %
%   O:0.0/6  MTR_OUT_BLT_REV  "Motor Starter OutFeed Belt Reverse VFD" %

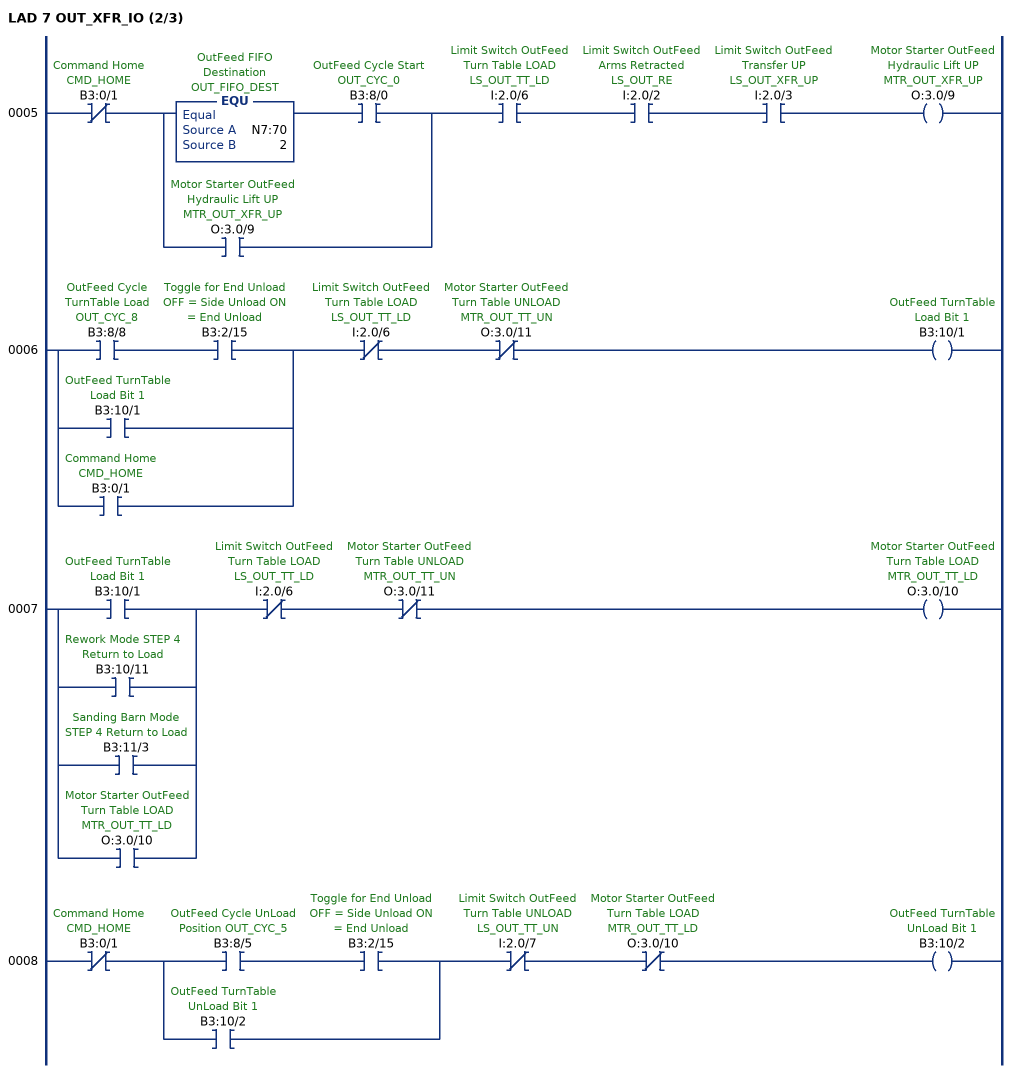
% Rung: 5 %
SOR XIO B3:0/1 BST EQU N7:70 2 XIC B3:8/0 NXB XIC O:3.0/9 BND XIC I:2.0/6 XIC I:2.0/2 XIC I:2.0/3 OTE O:3.0/9 EOR
%   B3:0/1  CMD_HOME  "Command Home" %
%   N7:70  OUT_FIFO_DEST  "OutFeed FIFO Destination" %
%   B3:8/0  OUT_CYC_0  "OutFeed Cycle Start" %
%   O:3.0/9  MTR_OUT_XFR_UP  "Motor Starter OutFeed Hydraulic Lift UP" %
%   I:2.0/6  LS_OUT_TT_LD  "Limit Switch OutFeed Turn Table LOAD" %
%   I:2.0/2  LS_OUT_RE  "Limit Switch OutFeed Arms Retracted" %
%   I:2.0/3  LS_OUT_XFR_UP  "Limit Switch OutFeed Transfer UP" %
% Rung: 6 %
SOR BST XIC B3:8/8 XIC B3:2/15 NXB XIC B3:10/1 NXB XIC B3:0/1 BND XIO I:2.0/6 XIO O:3.0/11 OTE B3:10/1 EOR
%   B3:8/8  OUT_CYC_8  "OutFeed Cycle TurnTable Load" %
%   B3:2/15  "Toggle for End Unload OFF = Side Unload ON = End Unload" %
%   B3:10/1  "OutFeed TurnTable Load Bit 1" %
%   B3:0/1  CMD_HOME  "Command Home" %
%   I:2.0/6  LS_OUT_TT_LD  "Limit Switch OutFeed Turn Table LOAD" %
%   O:3.0/11  MTR_OUT_TT_UN  "Motor Starter OutFeed Turn Table UNLOAD" %
% Rung: 7 %
SOR BST XIC B3:10/1 NXB XIC B3:10/11 NXB XIC B3:11/3 NXB XIC O:3.0/10 BND XIO I:2.0/6 XIO O:3.0/11 OTE O:3.0/10 EOR
%   B3:10/1  "OutFeed TurnTable Load Bit 1" %
%   B3:10/11  "Rework Mode STEP 4 Return to Load" %
%   B3:11/3  "Sanding Barn Mode STEP 4 Return to Load" %
%   O:3.0/10  MTR_OUT_TT_LD  "Motor Starter OutFeed Turn Table LOAD" %
%   I:2.0/6  LS_OUT_TT_LD  "Limit Switch OutFeed Turn Table LOAD" %
%   O:3.0/11  MTR_OUT_TT_UN  "Motor Starter OutFeed Turn Table UNLOAD" %
% Rung: 8 %
SOR XIO B3:0/1 BST XIC B3:8/5 XIC B3:2/15 NXB XIC B3:10/2 BND XIO I:2.0/7 XIO O:3.0/10 OTE B3:10/2 EOR
%   B3:0/1  CMD_HOME  "Command Home" %
%   B3:8/5  OUT_CYC_5  "OutFeed Cycle UnLoad Position" %
%   B3:2/15  "Toggle for End Unload OFF = Side Unload ON = End Unload" %
%   B3:10/2  "OutFeed TurnTable UnLoad Bit 1" %
%   I:2.0/7  LS_OUT_TT_UN  "Limit Switch OutFeed Turn Table UNLOAD" %
%   O:3.0/10  MTR_OUT_TT_LD  "Motor Starter OutFeed Turn Table LOAD" %

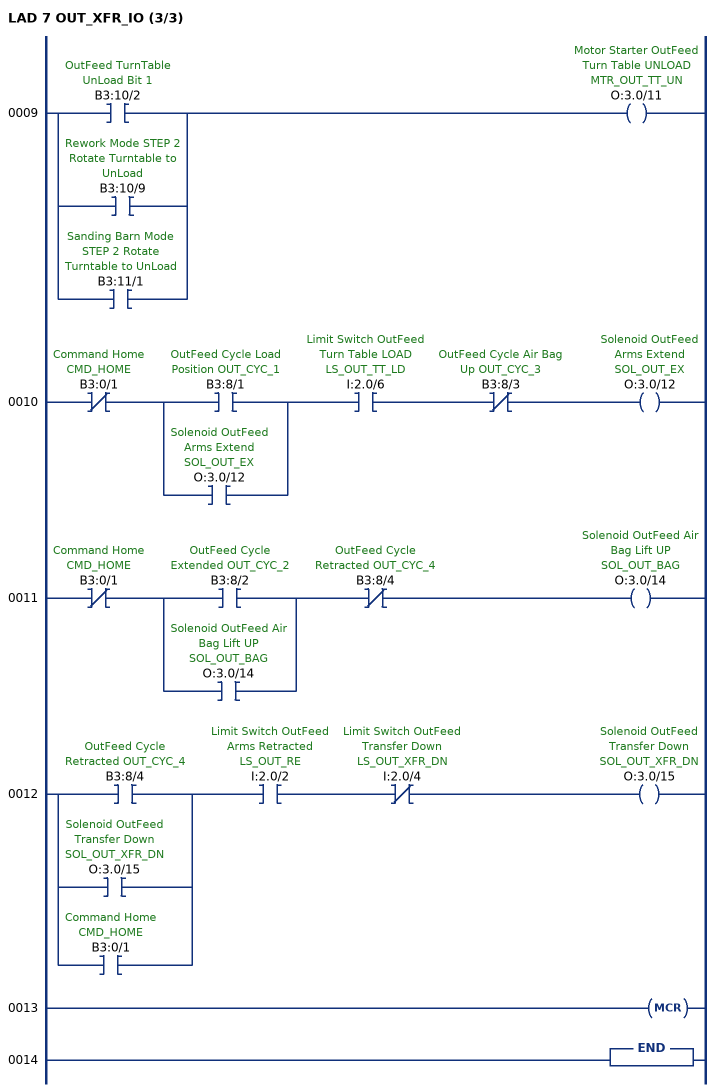
% Rung: 9 %
SOR BST XIC B3:10/2 NXB XIC B3:10/9 NXB XIC B3:11/1 BND OTE O:3.0/11 EOR
%   B3:10/2  "OutFeed TurnTable UnLoad Bit 1" %
%   B3:10/9  "Rework Mode STEP 2 Rotate Turntable to UnLoad" %
%   B3:11/1  "Sanding Barn Mode STEP 2 Rotate Turntable to UnLoad" %
%   O:3.0/11  MTR_OUT_TT_UN  "Motor Starter OutFeed Turn Table UNLOAD" %
% Rung: 10 %
SOR XIO B3:0/1 BST XIC B3:8/1 NXB XIC O:3.0/12 BND XIC I:2.0/6 XIO B3:8/3 OTE O:3.0/12 EOR
%   B3:0/1  CMD_HOME  "Command Home" %
%   B3:8/1  OUT_CYC_1  "OutFeed Cycle Load Position" %
%   O:3.0/12  SOL_OUT_EX  "Solenoid OutFeed Arms Extend" %
%   I:2.0/6  LS_OUT_TT_LD  "Limit Switch OutFeed Turn Table LOAD" %
%   B3:8/3  OUT_CYC_3  "OutFeed Cycle Air Bag Up" %
% Rung: 11 %
SOR XIO B3:0/1 BST XIC B3:8/2 NXB XIC O:3.0/14 BND XIO B3:8/4 OTE O:3.0/14 EOR
%   B3:0/1  CMD_HOME  "Command Home" %
%   B3:8/2  OUT_CYC_2  "OutFeed Cycle Extended" %
%   O:3.0/14  SOL_OUT_BAG  "Solenoid OutFeed Air Bag Lift UP" %
%   B3:8/4  OUT_CYC_4  "OutFeed Cycle Retracted" %
% Rung: 12 %
SOR BST XIC B3:8/4 NXB XIC O:3.0/15 NXB XIC B3:0/1 BND XIC I:2.0/2 XIO I:2.0/4 OTE O:3.0/15 EOR
%   B3:8/4  OUT_CYC_4  "OutFeed Cycle Retracted" %
%   O:3.0/15  SOL_OUT_XFR_DN  "Solenoid OutFeed Transfer Down" %
%   B3:0/1  CMD_HOME  "Command Home" %
%   I:2.0/2  LS_OUT_RE  "Limit Switch OutFeed Arms Retracted" %
%   I:2.0/4  LS_OUT_XFR_DN  "Limit Switch OutFeed Transfer Down" %
% Rung: 13 %
SOR MCR EOR
% Rung: 14 %
SOR END EOR

LADDER 8 "OUT_UNLOAD"    % OutFeed UnLoad Cycle %
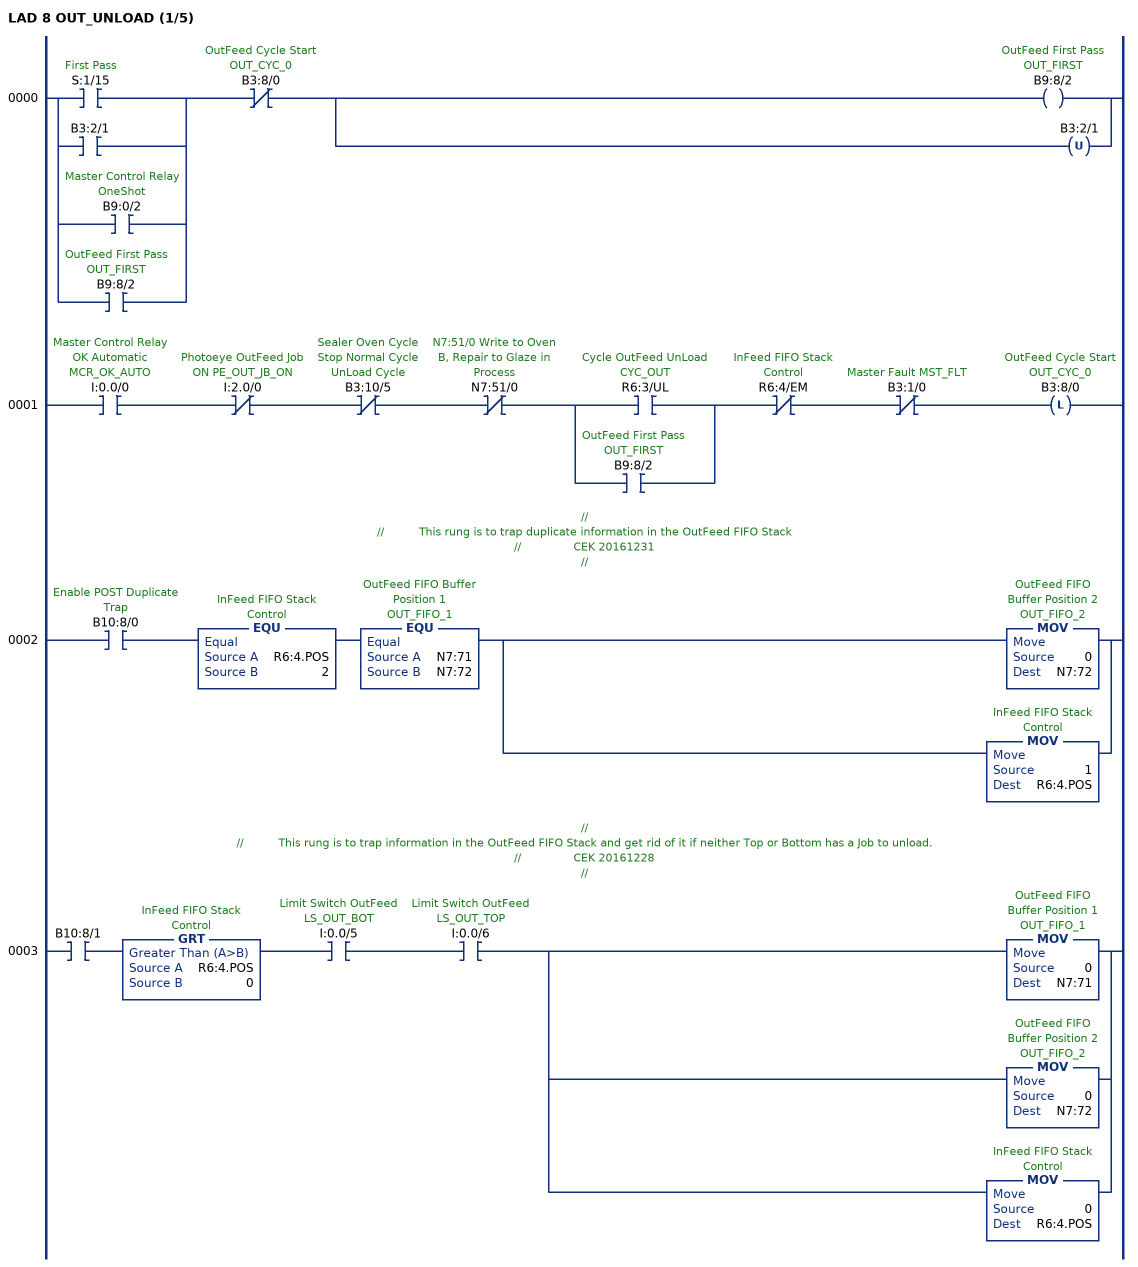
% Rung: 0 %
SOR BST XIC S:1/15 NXB XIC B3:2/1 NXB XIC B9:0/2 NXB XIC B9:8/2 BND XIO B3:8/0 BST OTE B9:8/2 NXB OTU B3:2/1 BND EOR
%   S:1/15  "First Pass" %
%   B9:0/2  "Master Control Relay OneShot" %
%   B9:8/2  OUT_FIRST  "OutFeed First Pass" %
%   B3:8/0  OUT_CYC_0  "OutFeed Cycle Start" %
% Rung: 1 %
SOR XIC I:0.0/0 XIO I:2.0/0 XIO B3:10/5 XIO N7:51/0 BST XIC R6:3/UL NXB XIC B9:8/2 BND XIO R6:4/EM XIO B3:1/0 OTL B3:8/0 EOR
%   I:0.0/0  MCR_OK_AUTO  "Master Control Relay OK Automatic" %
%   I:2.0/0  PE_OUT_JB_ON  "Photoeye OutFeed Job ON" %
%   B3:10/5  "Sealer Oven Cycle Stop Normal Cycle UnLoad Cycle" %
%   N7:51/0  "N7:51/0 Write to Oven B, Repair to Glaze in Process" %
%   R6:3/UL  CYC_OUT  "Cycle OutFeed UnLoad" %
%   B9:8/2  OUT_FIRST  "OutFeed First Pass" %
%   R6:4  "InFeed FIFO Stack Control" %
%   B3:1/0  MST_FLT  "Master Fault" %
%   B3:8/0  OUT_CYC_0  "OutFeed Cycle Start" %
% Rung: 2 %
% //
% //          This rung is to trap duplicate information in the OutFeed FIFO Stack
% //               CEK 20161231
% // %
SOR XIC B10:8/0 EQU R6:4.POS 2 EQU N7:71 N7:72 BST MOV 0 N7:72 NXB MOV 1 R6:4.POS BND EOR
%   B10:8/0  "Enable POST Duplicate Trap" %
%   R6:4  "InFeed FIFO Stack Control" %
%   N7:71  OUT_FIFO_1  "OutFeed FIFO Buffer Position 1" %
%   N7:72  OUT_FIFO_2  "OutFeed FIFO Buffer Position 2" %
% Rung: 3 %
% //
% //          This rung is to trap information in the OutFeed FIFO Stack and get rid of it if neither Top or Bottom has a Job to unload.
% //               CEK 20161228
% // %
SOR XIC B10:8/1 GRT R6:4.POS 0 XIC I:0.0/5 XIC I:0.0/6 BST MOV 0 N7:71 NXB MOV 0 N7:72 NXB MOV 0 R6:4.POS BND EOR
%   R6:4  "InFeed FIFO Stack Control" %
%   I:0.0/5  LS_OUT_BOT  "Limit Switch OutFeed" %
%   I:0.0/6  LS_OUT_TOP  "Limit Switch OutFeed" %
%   N7:71  OUT_FIFO_1  "OutFeed FIFO Buffer Position 1" %
%   N7:72  OUT_FIFO_2  "OutFeed FIFO Buffer Position 2" %

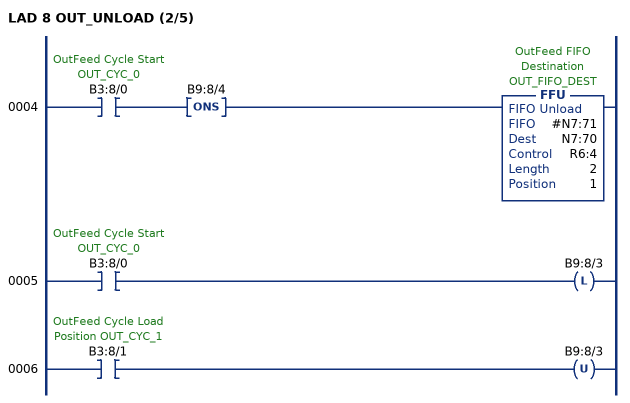
% Rung: 4 %
SOR XIC B3:8/0 ONS B9:8/4 FFU #N7:71 N7:70 R6:4 2 1 EOR
%   B3:8/0  OUT_CYC_0  "OutFeed Cycle Start" %
%   N7:71  OUT_FIFO_1  "OutFeed FIFO Buffer Position 1" %
%   N7:70  OUT_FIFO_DEST  "OutFeed FIFO Destination" %
%   R6:4  "InFeed FIFO Stack Control" %
% Rung: 5 %
SOR XIC B3:8/0 OTL B9:8/3 EOR
%   B3:8/0  OUT_CYC_0  "OutFeed Cycle Start" %
% Rung: 6 %
SOR XIC B3:8/1 OTU B9:8/3 EOR
%   B3:8/1  OUT_CYC_1  "OutFeed Cycle Load Position" %

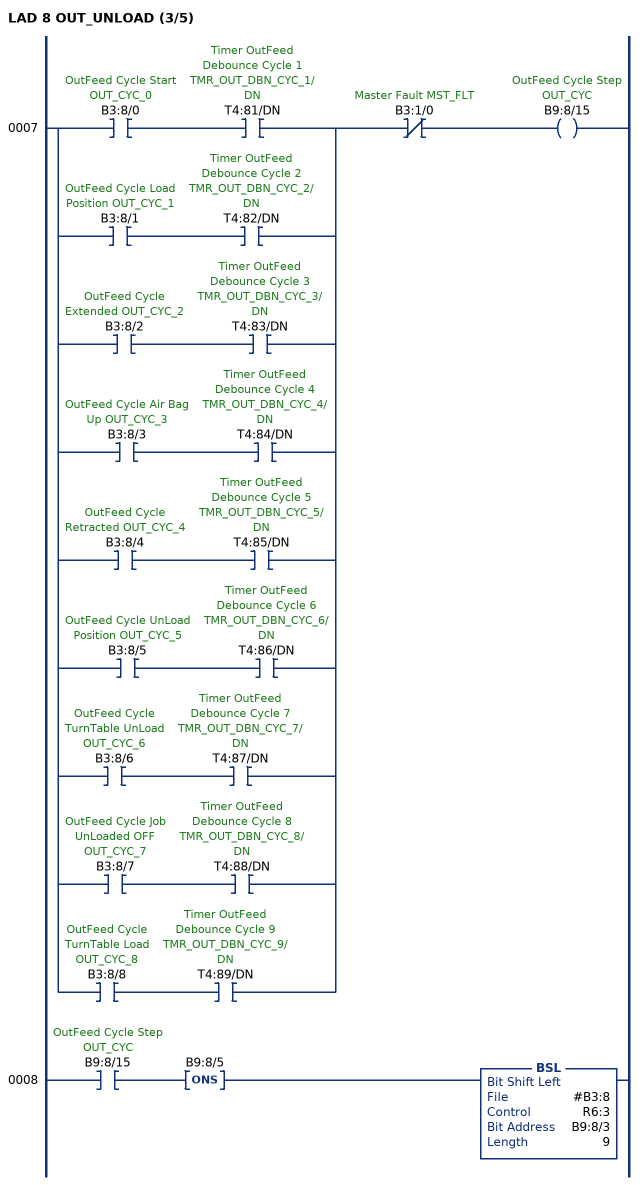
% Rung: 7 %
SOR BST XIC B3:8/0 XIC T4:81/DN NXB XIC B3:8/1 XIC T4:82/DN NXB XIC B3:8/2 XIC T4:83/DN NXB XIC B3:8/3 XIC T4:84/DN NXB XIC B3:8/4 XIC T4:85/DN NXB XIC B3:8/5 XIC T4:86/DN NXB XIC B3:8/6 XIC T4:87/DN NXB XIC B3:8/7 XIC T4:88/DN NXB XIC B3:8/8 XIC T4:89/DN BND XIO B3:1/0 OTE B9:8/15 EOR
%   B3:8/0  OUT_CYC_0  "OutFeed Cycle Start" %
%   T4:81  TMR_OUT_DBN_CYC_1  "Timer OutFeed Debounce Cycle 1" %
%   B3:8/1  OUT_CYC_1  "OutFeed Cycle Load Position" %
%   T4:82  TMR_OUT_DBN_CYC_2  "Timer OutFeed Debounce Cycle 2" %
%   B3:8/2  OUT_CYC_2  "OutFeed Cycle Extended" %
%   T4:83  TMR_OUT_DBN_CYC_3  "Timer OutFeed Debounce Cycle 3" %
%   B3:8/3  OUT_CYC_3  "OutFeed Cycle Air Bag Up" %
%   T4:84  TMR_OUT_DBN_CYC_4  "Timer OutFeed Debounce Cycle 4" %
%   B3:8/4  OUT_CYC_4  "OutFeed Cycle Retracted" %
%   T4:85  TMR_OUT_DBN_CYC_5  "Timer OutFeed Debounce Cycle 5" %
%   B3:8/5  OUT_CYC_5  "OutFeed Cycle UnLoad Position" %
%   T4:86  TMR_OUT_DBN_CYC_6  "Timer OutFeed Debounce Cycle 6" %
%   B3:8/6  OUT_CYC_6  "OutFeed Cycle TurnTable UnLoad" %
%   T4:87  TMR_OUT_DBN_CYC_7  "Timer OutFeed Debounce Cycle 7" %
%   B3:8/7  OUT_CYC_7  "OutFeed Cycle Job UnLoaded OFF" %
%   T4:88  TMR_OUT_DBN_CYC_8  "Timer OutFeed Debounce Cycle 8" %
%   B3:8/8  OUT_CYC_8  "OutFeed Cycle TurnTable Load" %
%   T4:89  TMR_OUT_DBN_CYC_9  "Timer OutFeed Debounce Cycle 9" %
%   B3:1/0  MST_FLT  "Master Fault" %
%   B9:8/15  OUT_CYC  "OutFeed Cycle Step" %
% Rung: 8 %
SOR XIC B9:8/15 ONS B9:8/5 BSL #B3:8 R6:3 B9:8/3 9 EOR
%   B9:8/15  OUT_CYC  "OutFeed Cycle Step" %

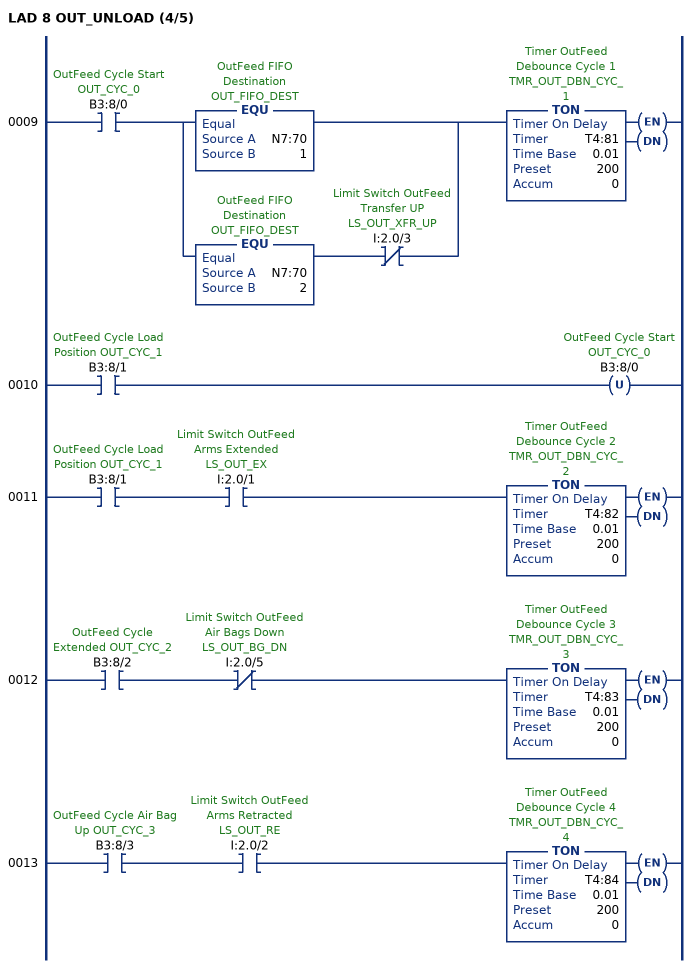
% Rung: 9 %
SOR XIC B3:8/0 BST EQU N7:70 1 NXB EQU N7:70 2 XIO I:2.0/3 BND TON T4:81 0.01 200 0 EOR
%   B3:8/0  OUT_CYC_0  "OutFeed Cycle Start" %
%   N7:70  OUT_FIFO_DEST  "OutFeed FIFO Destination" %
%   I:2.0/3  LS_OUT_XFR_UP  "Limit Switch OutFeed Transfer UP" %
%   T4:81  TMR_OUT_DBN_CYC_1  "Timer OutFeed Debounce Cycle 1" %
% Rung: 10 %
SOR XIC B3:8/1 OTU B3:8/0 EOR
%   B3:8/1  OUT_CYC_1  "OutFeed Cycle Load Position" %
%   B3:8/0  OUT_CYC_0  "OutFeed Cycle Start" %
% Rung: 11 %
SOR XIC B3:8/1 XIC I:2.0/1 TON T4:82 0.01 200 0 EOR
%   B3:8/1  OUT_CYC_1  "OutFeed Cycle Load Position" %
%   I:2.0/1  LS_OUT_EX  "Limit Switch OutFeed Arms Extended" %
%   T4:82  TMR_OUT_DBN_CYC_2  "Timer OutFeed Debounce Cycle 2" %
% Rung: 12 %
SOR XIC B3:8/2 XIO I:2.0/5 TON T4:83 0.01 200 0 EOR
%   B3:8/2  OUT_CYC_2  "OutFeed Cycle Extended" %
%   I:2.0/5  LS_OUT_BG_DN  "Limit Switch OutFeed Air Bags Down" %
%   T4:83  TMR_OUT_DBN_CYC_3  "Timer OutFeed Debounce Cycle 3" %
% Rung: 13 %
SOR XIC B3:8/3 XIC I:2.0/2 TON T4:84 0.01 200 0 EOR
%   B3:8/3  OUT_CYC_3  "OutFeed Cycle Air Bag Up" %
%   I:2.0/2  LS_OUT_RE  "Limit Switch OutFeed Arms Retracted" %
%   T4:84  TMR_OUT_DBN_CYC_4  "Timer OutFeed Debounce Cycle 4" %

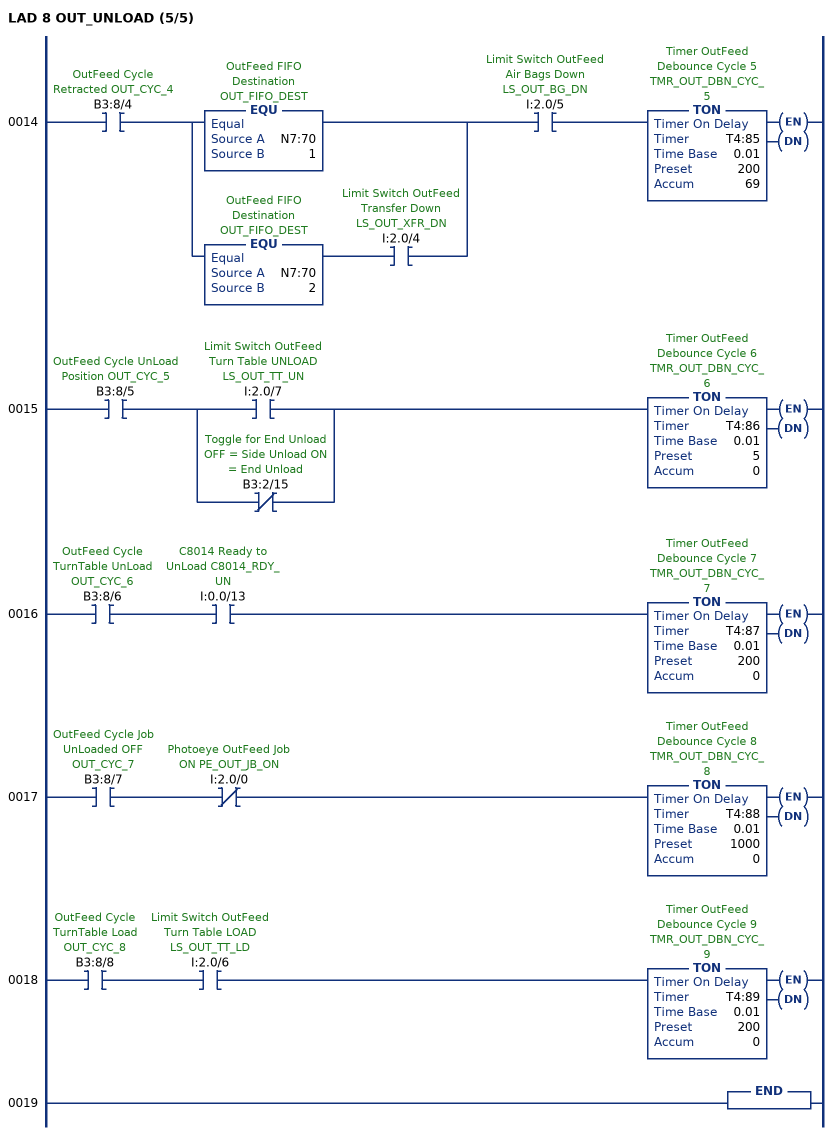
% Rung: 14 %
SOR XIC B3:8/4 BST EQU N7:70 1 NXB EQU N7:70 2 XIC I:2.0/4 BND XIC I:2.0/5 TON T4:85 0.01 200 69 EOR
%   B3:8/4  OUT_CYC_4  "OutFeed Cycle Retracted" %
%   N7:70  OUT_FIFO_DEST  "OutFeed FIFO Destination" %
%   I:2.0/4  LS_OUT_XFR_DN  "Limit Switch OutFeed Transfer Down" %
%   I:2.0/5  LS_OUT_BG_DN  "Limit Switch OutFeed Air Bags Down" %
%   T4:85  TMR_OUT_DBN_CYC_5  "Timer OutFeed Debounce Cycle 5" %
% Rung: 15 %
SOR XIC B3:8/5 BST XIC I:2.0/7 NXB XIO B3:2/15 BND TON T4:86 0.01 5 0 EOR
%   B3:8/5  OUT_CYC_5  "OutFeed Cycle UnLoad Position" %
%   I:2.0/7  LS_OUT_TT_UN  "Limit Switch OutFeed Turn Table UNLOAD" %
%   B3:2/15  "Toggle for End Unload OFF = Side Unload ON = End Unload" %
%   T4:86  TMR_OUT_DBN_CYC_6  "Timer OutFeed Debounce Cycle 6" %
% Rung: 16 %
SOR XIC B3:8/6 XIC I:0.0/13 TON T4:87 0.01 200 0 EOR
%   B3:8/6  OUT_CYC_6  "OutFeed Cycle TurnTable UnLoad" %
%   I:0.0/13  C8014_RDY_UN  "C8014 Ready to UnLoad" %
%   T4:87  TMR_OUT_DBN_CYC_7  "Timer OutFeed Debounce Cycle 7" %
% Rung: 17 %
SOR XIC B3:8/7 XIO I:2.0/0 TON T4:88 0.01 1000 0 EOR
%   B3:8/7  OUT_CYC_7  "OutFeed Cycle Job UnLoaded OFF" %
%   I:2.0/0  PE_OUT_JB_ON  "Photoeye OutFeed Job ON" %
%   T4:88  TMR_OUT_DBN_CYC_8  "Timer OutFeed Debounce Cycle 8" %
% Rung: 18 %
SOR XIC B3:8/8 XIC I:2.0/6 TON T4:89 0.01 200 0 EOR
%   B3:8/8  OUT_CYC_8  "OutFeed Cycle TurnTable Load" %
%   I:2.0/6  LS_OUT_TT_LD  "Limit Switch OutFeed Turn Table LOAD" %
%   T4:89  TMR_OUT_DBN_CYC_9  "Timer OutFeed Debounce Cycle 9" %
% Rung: 19 %
SOR END EOR

LADDER 10 "FLT"    % Operation Faults %
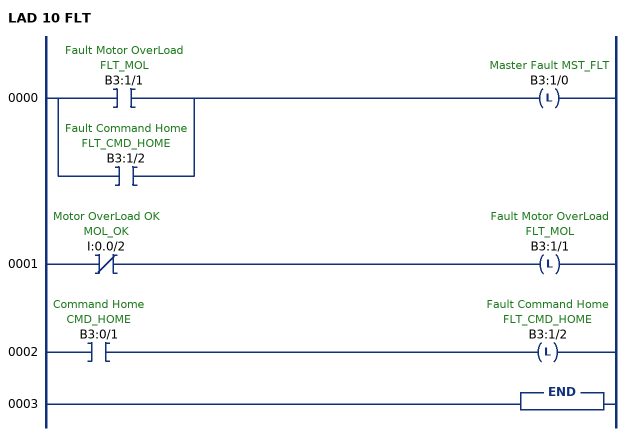
% Rung: 0 %
SOR BST XIC B3:1/1 NXB XIC B3:1/2 BND OTL B3:1/0 EOR
%   B3:1/1  FLT_MOL  "Fault Motor OverLoad" %
%   B3:1/2  FLT_CMD_HOME  "Fault Command Home" %
%   B3:1/0  MST_FLT  "Master Fault" %
% Rung: 1 %
SOR XIO I:0.0/2 OTL B3:1/1 EOR
%   I:0.0/2  MOL_OK  "Motor OverLoad OK" %
%   B3:1/1  FLT_MOL  "Fault Motor OverLoad" %
% Rung: 2 %
SOR XIC B3:0/1 OTL B3:1/2 EOR
%   B3:0/1  CMD_HOME  "Command Home" %
%   B3:1/2  FLT_CMD_HOME  "Fault Command Home" %
% Rung: 3 %
SOR END EOR

LADDER 11 "PTV"
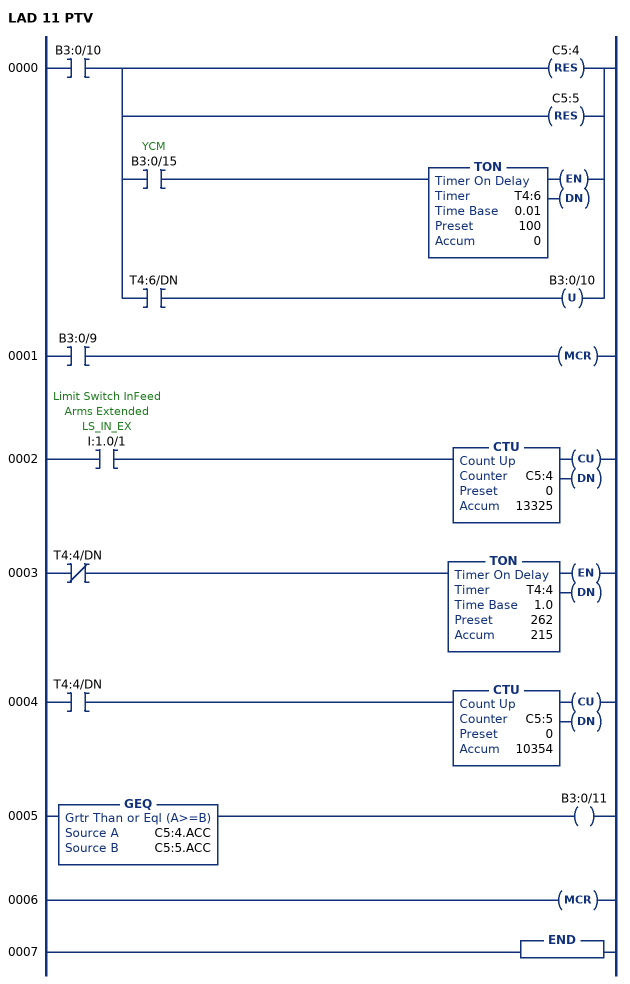
% Rung: 0 %
SOR XIC B3:0/10 BST RES C5:4 NXB RES C5:5 NXB XIC B3:0/15 TON T4:6 0.01 100 0 NXB XIC T4:6/DN OTU B3:0/10 BND EOR
%   B3:0/15  YCM %
% Rung: 1 %
SOR XIC B3:0/9 MCR EOR
% Rung: 2 %
SOR XIC I:1.0/1 CTU C5:4 0 13325 EOR
%   I:1.0/1  LS_IN_EX  "Limit Switch InFeed Arms Extended" %
% Rung: 3 %
SOR XIO T4:4/DN TON T4:4 1.0 262 215 EOR
% Rung: 4 %
SOR XIC T4:4/DN CTU C5:5 0 10354 EOR
% Rung: 5 %
SOR GEQ C5:4.ACC C5:5.ACC OTE B3:0/11 EOR
% Rung: 6 %
SOR MCR EOR
% Rung: 7 %
SOR END EOR

LADDER 12 "TOP COAT B"
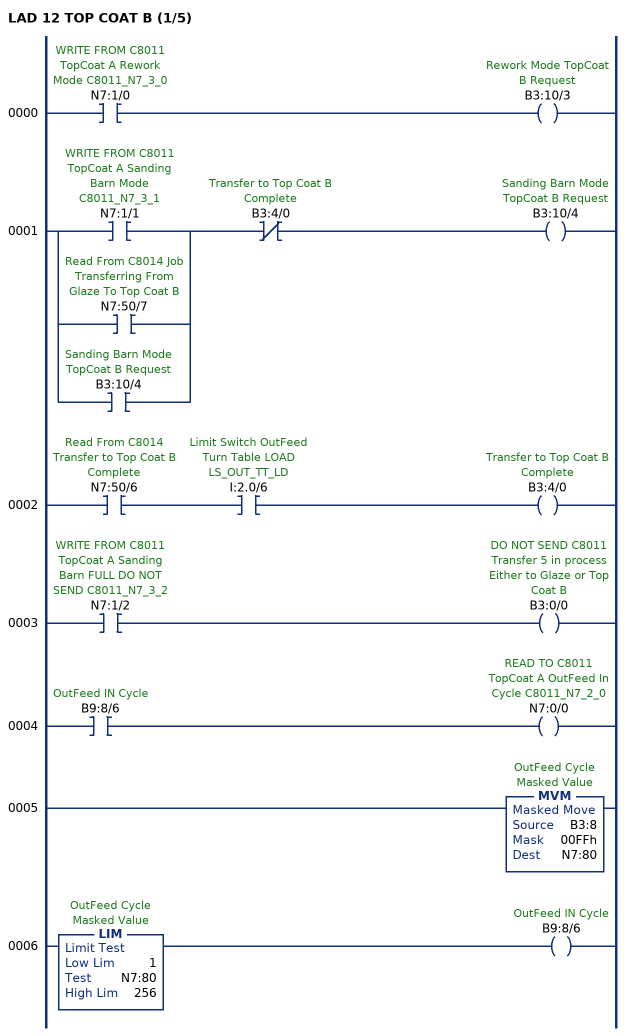
% Rung: 0 %
SOR XIC N7:1/0 OTE B3:10/3 EOR
%   N7:1/0  C8011_N7_3_0  "WRITE FROM C8011 TopCoat A Rework Mode" %
%   B3:10/3  "Rework Mode TopCoat B Request" %
% Rung: 1 %
SOR BST XIC N7:1/1 NXB XIC N7:50/7 NXB XIC B3:10/4 BND XIO B3:4/0 OTE B3:10/4 EOR
%   N7:1/1  C8011_N7_3_1  "WRITE FROM C8011 TopCoat A Sanding Barn Mode" %
%   N7:50/7  "Read From C8014 Job Transferring From Glaze To Top Coat B" %
%   B3:10/4  "Sanding Barn Mode TopCoat B Request" %
%   B3:4/0  "Transfer to Top Coat B Complete" %
% Rung: 2 %
SOR XIC N7:50/6 XIC I:2.0/6 OTE B3:4/0 EOR
%   N7:50/6  "Read From C8014 Transfer to Top Coat B Complete" %
%   I:2.0/6  LS_OUT_TT_LD  "Limit Switch OutFeed Turn Table LOAD" %
%   B3:4/0  "Transfer to Top Coat B Complete" %
% Rung: 3 %
SOR XIC N7:1/2 OTE B3:0/0 EOR
%   N7:1/2  C8011_N7_3_2  "WRITE FROM C8011 TopCoat A Sanding Barn FULL DO NOT SEND" %
%   B3:0/0  "DO NOT SEND C8011 Transfer 5 in process Either to Glaze or Top Coat B" %
% Rung: 4 %
SOR XIC B9:8/6 OTE N7:0/0 EOR
%   B9:8/6  "OutFeed IN Cycle" %
%   N7:0/0  C8011_N7_2_0  "READ TO C8011 TopCoat A OutFeed In Cycle" %
% Rung: 5 %
SOR MVM B3:8 00FFh N7:80 EOR
%   N7:80  "OutFeed Cycle Masked Value" %
% Rung: 6 %
SOR LIM 1 N7:80 256 OTE B9:8/6 EOR
%   N7:80  "OutFeed Cycle Masked Value" %
%   B9:8/6  "OutFeed IN Cycle" %

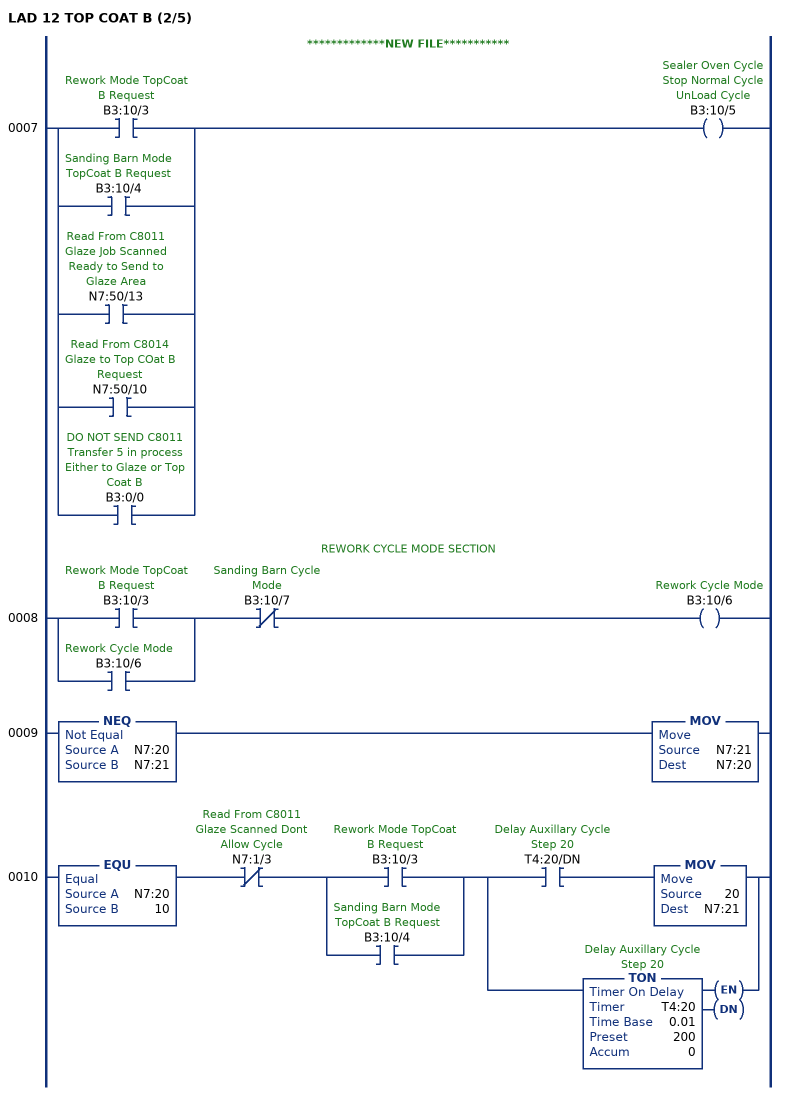
% Rung: 7 %
% TITLE: *************NEW FILE*********** %
SOR BST XIC B3:10/3 NXB XIC B3:10/4 NXB XIC N7:50/13 NXB XIC N7:50/10 NXB XIC B3:0/0 BND OTE B3:10/5 EOR
%   B3:10/3  "Rework Mode TopCoat B Request" %
%   B3:10/4  "Sanding Barn Mode TopCoat B Request" %
%   N7:50/13  "Read From C8011 Glaze Job Scanned Ready to Send to Glaze Area" %
%   N7:50/10  "Read From C8014 Glaze to Top COat B Request" %
%   B3:0/0  "DO NOT SEND C8011 Transfer 5 in process Either to Glaze or Top Coat B" %
%   B3:10/5  "Sealer Oven Cycle Stop Normal Cycle UnLoad Cycle" %
% Rung: 8 %
% REWORK CYCLE MODE SECTION %
SOR BST XIC B3:10/3 NXB XIC B3:10/6 BND XIO B3:10/7 OTE B3:10/6 EOR
%   B3:10/3  "Rework Mode TopCoat B Request" %
%   B3:10/6  "Rework Cycle Mode" %
%   B3:10/7  "Sanding Barn Cycle Mode" %
% Rung: 9 %
SOR NEQ N7:20 N7:21 MOV N7:21 N7:20 EOR
% Rung: 10 %
SOR EQU N7:20 10 XIO N7:1/3 BST XIC B3:10/3 NXB XIC B3:10/4 BND BST XIC T4:20/DN MOV 20 N7:21 NXB TON T4:20 0.01 200 0 BND EOR
%   N7:1/3  "Read From C8011 Glaze Scanned Dont Allow Cycle" %
%   B3:10/3  "Rework Mode TopCoat B Request" %
%   B3:10/4  "Sanding Barn Mode TopCoat B Request" %
%   T4:20  "Delay Auxillary Cycle Step 20" %

